// TIA Portal project "Inspection_system" (V16)

(* hardware
DEVICE "S71500/ET200MP station_1"  S7-1500 station
   slot 0: "Rail_0"  Rack  6ES7 590-1***0-0AA0
   slot 1: "PLC_1"  CPU 1515-2 PN  6ES7 515-2AM01-0AB0  V2.8
      slot 3: "CPU display_1"  6ES7591-1BA00-0AA0
      slot 32768: "PROFINET interface_1"  X1
         slot 32769: "Port_1"  X1 P1
         slot 32770: "Port_2"  X1 P2
      slot 33024: "PROFINET interface_2"  X2
         slot 33025: "Port_1"  X2 P1
      slot 34817: "Virtual CP interface port_1"  Virtual CP interface port  Virtual CP interface port
DEVICE "ET 200SP station_1"  ET 200SP-Station
   slot 0: "Rack_0"  Rack  6ES5 710-8MAx1
   slot 0: "IO device_1"  IM 155-6 PN/2 HF  6ES7 155-6AU01-0CN0  V4.2
   slot 1: "AI 4xRTD/TC 2-,3-,4-wire HF_1"  AI 4xRTD/TC 2-,3-,4-wire HF  6ES7 134-6JD00-0CA1  V2.0
      slot 1: "AI 4xRTD/TC 2-,3-,4-wire HF_1"  AI 4xRTD/TC 2-,3-,4-wire HF
   slot 2: "AI 4xRTD/TC 2-,3-,4-wire HF_2"  AI 4xRTD/TC 2-,3-,4-wire HF  6ES7 134-6JD00-0CA1  V2.0
      slot 1: "AI 4xRTD/TC 2-,3-,4-wire HF_2"  AI 4xRTD/TC 2-,3-,4-wire HF
   slot 3: "AI 4xRTD/TC 2-,3-,4-wire HF_3"  AI 4xRTD/TC 2-,3-,4-wire HF  6ES7 134-6JD00-0CA1  V2.0
      slot 1: "AI 4xRTD/TC 2-,3-,4-wire HF_3"  AI 4xRTD/TC 2-,3-,4-wire HF
   slot 4: "AI 8xI 2-,4-wire BA_1"  AI 8xI 2-,4-wire BA  6ES7 134-6GF00-0AA1  V1.0
      slot 1: "AI 8xI 2-,4-wire BA_1"  AI 8xI 2-,4-wire BA
   slot 5: "AQ 4xU/I ST_1"  AQ 4xU/I ST  6ES7 135-6HD00-0BA1  V1.1
      slot 1: "AQ 4xU/I ST_1"  AQ 4xU/I ST
   slot 6: "AQ 4xU/I ST_2"  AQ 4xU/I ST  6ES7 135-6HD00-0BA1  V1.1
      slot 1: "AQ 4xU/I ST_2"  AQ 4xU/I ST
   slot 7: "AQ 4xU/I ST_3"  AQ 4xU/I ST  6ES7 135-6HD00-0BA1  V1.1
      slot 1: "AQ 4xU/I ST_3"  AQ 4xU/I ST
   slot 8: "AQ 4xU/I ST_4"  AQ 4xU/I ST  6ES7 135-6HD00-0BA1  V1.1
      slot 1: "AQ 4xU/I ST_4"  AQ 4xU/I ST
   slot 9: "AQ 4xU/I ST_5"  AQ 4xU/I ST  6ES7 135-6HD00-0BA1  V1.1
      slot 1: "AQ 4xU/I ST_5"  AQ 4xU/I ST
   slot 10: "AQ 4xU/I ST_6"  AQ 4xU/I ST  6ES7 135-6HD00-0BA1  V1.1
      slot 1: "AQ 4xU/I ST_6"  AQ 4xU/I ST
   slot 11: "AQ 4xU/I ST_7"  AQ 4xU/I ST  6ES7 135-6HD00-0BA1  V1.1
      slot 1: "AQ 4xU/I ST_7"  AQ 4xU/I ST
   slot 12: "AQ 4xU/I ST_8"  AQ 4xU/I ST  6ES7 135-6HD00-0BA1  V1.1
      slot 1: "AQ 4xU/I ST_8"  AQ 4xU/I ST
   slot 13: "DI 16x24VDC ST_1"  DI 16x24VDC ST  6ES7 131-6BH01-0BA0  V0.0
      slot 1: "DI 16x24VDC ST_1"  DI 16x24VDC ST
   slot 14: "DQ 16x24VDC/0.5A ST_1"  DQ 16x24VDC/0.5A ST  6ES7 132-6BH01-0BA0  V0.0
      slot 1: "DQ 16x24VDC/0.5A ST_1"  DQ 16x24VDC/0.5A ST
   slot 15: "DQ 16x24VDC/0.5A ST_2"  DQ 16x24VDC/0.5A ST  6ES7 132-6BH01-0BA0  V0.0
      slot 1: "DQ 16x24VDC/0.5A ST_2"  DQ 16x24VDC/0.5A ST
   slot 16: "Server module_1"  Server module  6ES7 193-6PA00-0AA0  V1.1
      slot 1: "Server module_1"  Server module
   slot 127: "BA 2xRJ45"  BA 2xRJ45  6ES7 193-6AR00-0AA0  V0.0
      slot 1: "Port_1"  X1 P1 R  6ES7 193-6AR00-0AA0  V0.0
      slot 2: "Port_2"  X1 P2 R  6ES7 193-6AR00-0AA0  V0.0
*)

// ===== PLC "PLC_1"  CPU 1515-2 PN =====

VAR_GLOBAL   // PLC tag table "Default tag table"
   "upTempLaser1" AT %IW42 : Int;   // (Ain0.0)
   "upTempLaser2" AT %IW44 : Int;   // (Ain0.1)
   "upTempCam1" AT %IW46 : Int;   // (Ain0.2)
   "upTempCam2" AT %IW48 : Int;   // (Ain0.3)
   "downTempLaser1" AT %IW8 : Int;   // (Ain0.4)
   "downTempLaser2" AT %IW10 : Int;   // (Ain0.5)
   "downTempCam1" AT %IW12 : Int;   // (Ain0.6)
   "downTempCam2" AT %IW14 : Int;   // (Ain0.7)
   "airTemperatur" AT %IW16 : Int;   // (Ain1.0)
   "speedRaw" AT %IW24 : Int;   // (Ain2.0)
   "upBlue1" AT %QW0 : Int;
   "upBlue2" AT %QW2 : Int;
   "upBlue3" AT %QW4 : Int;
   "upGreen1" AT %QW6 : Int;
   "upGreen2" AT %QW8 : Int;
   "upGreen3" AT %QW10 : Int;
   "upBlue4" AT %QW12 : Int;
   "upBlue5" AT %QW14 : Int;
   "upBlue6" AT %QW16 : Int;
   "upGreen4" AT %QW18 : Int;
   "upGreen5" AT %QW20 : Int;
   "upGreen6" AT %QW22 : Int;
   "upBlue7" AT %QW24 : Int;
   "upBlue8" AT %QW26 : Int;
   "upBlue9" AT %QW28 : Int;
   "downGreen1" AT %QW32 : Int;
   "downGreen2" AT %QW34 : Int;
   "downGreen3" AT %QW36 : Int;
   "downBlue1" AT %QW38 : Int;
   "downBlue2" AT %QW40 : Int;
   "downBlue3" AT %QW42 : Int;
   "downGreen4" AT %QW44 : Int;
   "downGreen5" AT %QW46 : Int;
   "downGreen6" AT %QW48 : Int;
   "downBlue4" AT %QW50 : Int;
   "downBlue5" AT %QW52 : Int;
   "downBlue6" AT %QW54 : Int;
   "downGreen7" AT %QW56 : Int;
   "downGreen8" AT %QW58 : Int;
   "downGreen9" AT %QW60 : Int;
   "door1" AT %I40.0 : Bool;   // Дверь-1
   "door2" AT %I40.1 : Bool;   // Дверь-2
   "power1_1Ok" AT %I40.2 : Bool;   // Питание внешних цепей
   "power1_2Ok" AT %I40.3 : Bool;   // Питание внутренних цепей
   "laserModeManual" AT %I40.6 : Bool;   // Режим лазеров - Ручной
   "laserModeAuto" AT %I40.7 : Bool;   // Режим лазеров - Автомат
   "veloModeManual" AT %I40.4 : Bool;   // Режим велосиметра - Ручной
   "veloModeAuto" AT %I40.5 : Bool;   // Режим велосиметра - Автомат
   "runForward" AT %I41.0 : Bool;   // Сигнал с цеха -- движение прямо
   "runBackward" AT %I41.1 : Bool;   // Сигнал с цеха -- движение обратно
   "resetAlm" AT %I41.2 : Bool;   // от кнопки сброса аварийного триггера
   "power2_1Ok" AT %I41.3 : Bool;   // Резервированный БП 2_2. Шкаф видеоинспекции, синхробокс и лазеры.
   "power2_2Ok" AT %I41.4 : Bool;   // Резервированный 2_1. Шкаф видеоинспекции, синхробокс и лазеры.
   "upBlue123" AT %Q64.0 : Bool;   // Включение синих лазеров BR1.1-BR1.3. Верх
   "upGreen123" AT %Q64.1 : Bool;   // Включение зелёных лазеров BR2.1-BR2.3. Верх
   "upBlue456" AT %Q64.2 : Bool;   // Включение синих лазеров BR3.1-BR3.3. Верх
   "upGreen456" AT %Q64.3 : Bool;   // Включение зелёных лазеров BR4.1-BR4.3. Верх
   "upBlue789" AT %Q64.4 : Bool;   // Включение синих лазеров BR5.1-BR5.3. Верх
   "downGreen123" AT %Q64.5 : Bool;   // Включение зелёных лазеров BR6.1-BR6.3. Низ
   "downBlue123" AT %Q64.6 : Bool;   // Включение синих лазеров BR7.1-BR7.3. Низ
   "downGreen465" AT %Q64.7 : Bool;   // Включение зелёных лазеров BR8.1-BR8.3. Низ
   "downBlue456" AT %Q65.0 : Bool;   // Включение синих лазеров BR9.1-BR9.3. Низ
   "downGreen789" AT %Q65.1 : Bool;   // Включение зелёных лазеров BR10.1-BR10.3. Низ
   "enLaserVelo" AT %Q66.0 : Bool;   // Лазер велосиметра
   "enGaugeVelo" AT %Q66.1 : Bool;   // Шторка затвора велосиметра
   "airClean" AT %Q66.2 : Bool;   // Клапан воздушного обдува (чистка стекол)
   "runSynchro" AT %Q66.3 : Bool;   // Пуск синхронизации
   "coolUpLaser" AT %Q66.4 : Bool;   // Вентиляторы верхних лазеров
   "coolUpCam" AT %Q66.5 : Bool;   // Вентилятор верхних камер
   "coolDownLaser" AT %Q66.6 : Bool;   // Вентиляторы нижних лазеров
   "coolDownCam" AT %Q66.7 : Bool;   // Вентилятор нижних камер
   "redLamp" AT %Q67.0 : Bool;   // Статус "Работа". Красная лампа.
   "greenLamp" AT %Q67.1 : Bool;   // Статус "Установка отключена". Зелёная лампа.
   "allCooling" AT %Q67.2 : Bool;   // Включение охладителя
   "reverse" AT %Q67.3 : Bool;   // Обратный ход линии
   "Tag_1" AT %M20.0 : Bool;
   "Tag_2" AT %M20.1 : Bool;
   "Tag_3" AT %M20.2 : Bool;
   "System_Byte" AT %MB1 : Byte;
   "FirstScan" AT %M1.0 : Bool;
   "DiagStatusUpdate" AT %M1.1 : Bool;
   "AlwaysTRUE" AT %M1.2 : Bool;
   "AlwaysFALSE" AT %M1.3 : Bool;
   "Clock_Byte" AT %MB0 : Byte;
   "Clock_10Hz" AT %M0.0 : Bool;
   "Clock_5Hz" AT %M0.1 : Bool;
   "Clock_2.5Hz" AT %M0.2 : Bool;
   "Clock_2Hz" AT %M0.3 : Bool;
   "Clock_1.25Hz" AT %M0.4 : Bool;
   "Clock_1Hz" AT %M0.5 : Bool;
   "Clock_0.625Hz" AT %M0.6 : Bool;
   "Clock_0.5Hz" AT %M0.7 : Bool;
END_VAR

DATA_BLOCK "Main_PRG"   // DB4
{ S7_Optimized_Access := 'TRUE' }
VERSION : 0.1
   VAR RETAIN
      AinOffset : Struct
         upTempLaser1 : Real;
         upTempLaser2 : Real;
         upTempCam1 : Real;
         upTempCam2 : Real;
         downTempLaser1 : Real;
         downTempLaser2 : Real;
         downTempCam1 : Real;
         downTempCam2 : Real;
         airTemperatur : Real;
         speed : Real;
      END_STRUCT;
   END_VAR
   VAR
      Ainputs : Struct
         upTempLaser1 : Real;
         upTempLaser2 : Real;
         upTempCam1 : Real;
         upTempCam2 : Real;
         downTempLaser1 : Real;
         downTempLaser2 : Real;
         downTempCam1 : Real;
         downTempCam2 : Real;
         airTemperatur : Real;
         speed : Real;
      END_STRUCT;
      fault_buffer : Struct   // 64bit -- Биты аварий
         door1 : Bool;   // Дверь1 -- открыта
         door2 : Bool;   // Дверь2 -- открыта
         power11 : Bool;   // Питание внешних цепей
         power12 : Bool;   // Питание внутренних цепей
         power2 : Bool;   // Питание лазеров, ШВИ, синхробокса, видеокамер
         upLaserTemp : Bool;   // Температура выше аварийного уровня. (Верхний блок лазеров)
         upLaserAllCh : Bool;   // Все каналы измерения температуры неисправны. (Верхний блок лазеров)
         upCamTemp : Bool;   // Температура выше аварийного уровня. (Верхний блок камер)
         upCamAllCh : Bool;   // Все каналы измерения температуры неисправны. (Верхний блок камер)
         downLaserTemp : Bool;   // Температура выше аварийного уровня. (Нижний блок лазеров)
         downLaserAllCh : Bool;   // Все каналы измерения температуры неисправны. (Нижний блок лазеров)
         downCamTemp : Bool;   // Температура выше аварийного уровня. (Нижний блок камер)
         downCamAllCh : Bool;   // Все каналы измерения температуры неисправны. (Нижний блок камер)
         Ain2MinLimit : Bool;   // Вход от велосиметра (4-20мА) ниже уровня 4мА
         Ain2MaxLimit : Bool;   // Вход от велосиметра (4-20мА) выше уровня 20мА
         iniError : Bool;   // Ошибка инициализации.
         gaugeOk : Bool;
         lasTempH : Bool := false;
         lasTempL : Bool := false;
         caseTempH : Bool := false;
         caseTempL : Bool := false;
         gaugeH : Bool := false;
         veloNoConnect : Bool;
         reserve7 : Bool := false;
         reserve8 : Bool := false;
         reserve9 : Bool := false;
         reserve10 : Bool := false;
         reserve11 : Bool := false;
         reserve12 : Bool := false;
         reserve13 : Bool := false;
         reserve14 : Bool := false;
         reserve15 : Bool := false;
         reserve16 : Bool := false;
         reserve17 : Bool := false;
         reserve18 : Bool := false;
         reserve19 : Bool := false;
         reserve20 : Bool := false;
         reserve21 : Bool := false;
         reserve22 : Bool := false;
         reserve23 : Bool := false;
         reserve24 : Bool := false;
         reserve25 : Bool := false;
         reserve26 : Bool := false;
         reserve27 : Bool := false;
         reserve28 : Bool := false;
         reserve29 : Bool := false;
         reserve30 : Bool := false;
         reserve31 : Bool := false;
      END_STRUCT;
      iniOk : Bool;
      initializing : Bool;
      RUN : Bool;
      errUpTempLaser1 : Bool;   // (Ain0.0)
      errUpTempLaser2 : Bool;   // (Ain0.1)
      errUpTempCam1 : Bool;   // (Ain0.2)
      errUpTempCam2 : Bool;   // (Ain0.3)
      errDownTempLaser1 : Bool;   // (Ain0.4)
      errDownTempLaser2 : Bool;   // (Ain0.5)
      errDownTempCam1 : Bool;   // (Ain0.6)
      errDownTempCam2 : Bool;   // (Ain0.7)
      errAirTemperatur : Bool;   // (Ain1.0)
      synchroOn : Bool;
      t0 : Bool;
      t1 : Bool := false;
      t2 : Bool := false;
      t3 : Bool := false;
      t4 : Bool := false;
      t5 : Bool := false;
      configAI0 : Struct
         modulInfo0 : Byte;   // версия
         modulInfo1 : Byte;   // Количество структур следующих параметров
         modulInfo2 : Byte;   // Количество следующих блоков параметров модуля
         modulInfo3 : Byte;   // длина блока параметров модуля
         modulParam4 : Byte;   // bit0 -- Отсутствует напряжение питания.
         modulParam5 : Byte := 16#0;   // резерв
         modulParam6 : Byte := 16#0;
         modulParam7 : Byte := 16#0;
         modulParam8 : Byte := 16#0;
         modulParam9 : Byte := 16#0;
         channelInfo10 : Byte;   // количество следующих блоков параметров канала
         channelInfo11 : Byte := 16#0;   // Длина блока параметров канала
         "0channel0_12" : Byte;   // Тип измерения
         "1channel0_13" : Byte := 16#0;   // Диапазон измерений
         "2channel0_14" : Byte := 16#0;   // Температурный коэффициент
         "3channel0_15" : Byte := 16#0;   // Сглаживание
         "4channel0_16" : Byte := 16#0;   // Единица измерения и тип подключения
         "5channel0_17" : Byte := 16#0;   // бит4 - превышен лимит2, бит5 - ниже лимита2, бит6 - превышен лимит1, бит7 - ниже лимита1
         "6channel0_18" : Byte := 16#0;   // бит1-общий режим, бит2-короткое замыкание, бит4-обрыв, бит5-компенсация, бит6-ниже, бит7-выше
         "7channel0_19" : Byte := 16#0;   // резерв
         "8channel0_20" : Byte := 16#0;   // резерв
         "9channel0_21" : Byte := 16#0;   // резерв
         "10channel0_22" : Byte := 16#0;   // hardware interrupt1, high limit, byte0
         "11channel0_23" : Byte := 16#0;   // hardware interrupt1, high limit, byte1
         "12channel0_24" : Byte := 16#0;   // hardware interrupt1, low limit, byte0
         "13channel0_25" : Byte := 16#0;   // hardware interrupt1, low limit, byte1
         "14channel0_26" : Byte := 16#0;   // hardware interrupt2, high limit, byte0
         "15channel0_27" : Byte := 16#0;   // hardware interrupt2, high limit, byte1
         "16channel0_28" : Byte := 16#0;   // hardware interrupt2, low limit, byte0
         "17channel0_29" : Byte := 16#0;   // hardware interrupt2, low limit, byte1
         "18channel0_30" : Byte := 16#0;   // сопротивление, byte0
         "19channel0_31" : Byte := 16#0;   // сопротивление, byte1
         "20channel0_32" : Byte := 16#0;   // резерв
         "21channel0_33" : Byte := 16#0;   // резерв
         "0channel1_34" : Byte := 16#0;   // Тип измерения
         "1channel1_35" : Byte := 16#0;   // Диапазон измерений
         "2channel1_36" : Byte := 16#0;   // Температурный коэффициент
         "3channel1_37" : Byte := 16#0;   // Сглаживание
         "4channel1_38" : Byte := 16#0;   // Единица измерения и тип подключения
         "5channel1_39" : Byte := 16#0;   // бит4 - превышен лимит2, бит5 - ниже лимита2, бит6 - превышен лимит1, бит7 - ниже лимита1
         "6channel1_40" : Byte := 16#0;   // бит1-общий режим, бит2-короткое замыкание, бит4-обрыв, бит5-компенсация, бит6-ниже, бит7-выше
         "7channel1_41" : Byte := 16#0;   // резерв
         "8channel1_42" : Byte := 16#0;   // резерв
         "9channel1_43" : Byte := 16#0;   // резерв
         "10channel1_44" : Byte := 16#0;   // hardware interrupt1, high limit, byte0
         "11channel1_45" : Byte := 16#0;   // hardware interrupt1, high limit, byte1
         "12channel1_46" : Byte := 16#0;   // hardware interrupt1, low limit, byte0
         "13channel1_47" : Byte := 16#0;   // hardware interrupt1, low limit, byte1
         "14channel1_48" : Byte := 16#0;   // hardware interrupt2, high limit, byte0
         "15channel1_49" : Byte := 16#0;   // hardware interrupt2, high limit, byte1
         "16channel1_50" : Byte := 16#0;   // hardware interrupt2, low limit, byte0
         "17channel1_51" : Byte := 16#0;   // hardware interrupt2, low limit, byte1
         "18channel1_52" : Byte := 16#0;   // сопротивление, byte0
         "19channel1_53" : Byte := 16#0;   // сопротивление, byte1
         "20channel1_54" : Byte := 16#0;   // резерв
         "21channel1_55" : Byte := 16#0;   // резерв
         "0channel2_56" : Byte := 16#0;   // Тип измерения
         "1channel2_57" : Byte := 16#0;   // Диапазон измерений
         "2channel2_58" : Byte := 16#0;   // Температурный коэффициент
         "3channel2_59" : Byte := 16#0;   // Сглаживание
         "4channel2_60" : Byte := 16#0;   // Единица измерения и тип подключения
         "5channel2_61" : Byte := 16#0;   // бит4 - превышен лимит2, бит5 - ниже лимита2, бит6 - превышен лимит1, бит7 - ниже лимита1
         "6channel2_62" : Byte := 16#0;   // бит1-общий режим, бит2-короткое замыкание, бит4-обрыв, бит5-компенсация, бит6-ниже, бит7-выше
         "7channel2_63" : Byte := 16#0;   // резерв
         "8channel2_64" : Byte := 16#0;   // резерв
         "9channel2_65" : Byte := 16#0;   // резерв
         "10channel2_66" : Byte := 16#0;   // hardware interrupt1, high limit, byte0
         "11channel2_67" : Byte := 16#0;   // hardware interrupt1, high limit, byte1
         "12channel2_68" : Byte := 16#0;   // hardware interrupt1, low limit, byte0
         "13channel2_69" : Byte := 16#0;   // hardware interrupt1, low limit, byte1
         "14channel2_70" : Byte := 16#0;   // hardware interrupt2, high limit, byte0
         "15channel2_71" : Byte := 16#0;   // hardware interrupt2, high limit, byte1
         "16channel2_72" : Byte := 16#0;   // hardware interrupt2, low limit, byte0
         "17channel2_73" : Byte := 16#0;   // hardware interrupt2, low limit, byte1
         "18channel2_74" : Byte := 16#0;   // сопротивление, byte0
         "19channel2_75" : Byte := 16#0;   // сопротивление, byte1
         "20channel2_76" : Byte := 16#0;   // резерв
         "21channel2_77" : Byte := 16#0;   // резерв
         "0channel3_78" : Byte := 16#0;   // Тип измерения
         "1channel3_79" : Byte := 16#0;   // Диапазон измерений
         "2channel3_80" : Byte := 16#0;   // Температурный коэффициент
         "3channel3_81" : Byte := 16#0;   // Сглаживание
         "4channel3_82" : Byte := 16#0;   // Единица измерения и тип подключения
         "5channel3_83" : Byte := 16#0;   // бит4 - превышен лимит2, бит5 - ниже лимита2, бит6 - превышен лимит1, бит7 - ниже лимита1
         "6channel3_84" : Byte := 16#0;   // бит1-общий режим, бит2-короткое замыкание, бит4-обрыв, бит5-компенсация, бит6-ниже, бит7-выше
         "7channel3_85" : Byte := 16#0;   // резерв
         "8channel3_86" : Byte := 16#0;   // резерв
         "9channel3_87" : Byte := 16#0;   // резерв
         "10channel3_88" : Byte := 16#0;   // hardware interrupt1, high limit, byte0
         "11channel3_89" : Byte := 16#0;   // hardware interrupt1, high limit, byte1
         "12channel3_90" : Byte := 16#0;   // hardware interrupt1, low limit, byte0
         "13channel3_91" : Byte := 16#0;   // hardware interrupt1, low limit, byte1
         "14channel3_92" : Byte := 16#0;   // hardware interrupt2, high limit, byte0
         "15channel3_93" : Byte := 16#0;   // hardware interrupt2, high limit, byte1
         "16channel3_94" : Byte := 16#0;   // hardware interrupt2, low limit, byte0
         "17channel3_95" : Byte := 16#0;   // hardware interrupt2, low limit, byte1
         "18channel3_96" : Byte := 16#0;   // сопротивление, byte0
         "19channel3_97" : Byte := 16#0;   // сопротивление, byte1
         "20channel3_98" : Byte := 16#0;   // резерв
         "21channel3_99" : Byte := 16#0;   // резерв
      END_STRUCT;
   END_VAR
BEGIN
END_DATA_BLOCK

DATA_BLOCK "READ"   // DB200
{ S7_Optimized_Access := 'FALSE' }
VERSION : 0.1
   VAR
      fault : Struct   // 64bit -- Биты аварий
         door1 : Bool;   // Дверь1 -- открыта
         door2 : Bool;   // Дверь2 -- открыта
         power11 : Bool;   // Питание внешних цепей
         power12 : Bool;   // Питание внутренних цепей
         power2 : Bool;   // Питание лазеров, ШВИ, синхробокса, видеокамер
         upLaserTemp : Bool;   // Температура выше аварийного уровня. (Верхний блок лазеров)
         upLaserAllCh : Bool;   // Все каналы измерения температуры неисправны. (Верхний блок лазеров)
         upCamTemp : Bool;   // Температура выше аварийного уровня. (Верхний блок камер)
         upCamAllCh : Bool;   // Все каналы измерения температуры неисправны. (Верхний блок камер)
         downLaserTemp : Bool;   // Температура выше аварийного уровня. (Нижний блок лазеров)
         downLaserAllCh : Bool;   // Все каналы измерения температуры неисправны. (Нижний блок лазеров)
         downCamTemp : Bool;   // Температура выше аварийного уровня. (Нижний блок камер)
         downCamAllCh : Bool;   // Все каналы измерения температуры неисправны. (Нижний блок камер)
         Ain2MinLimit : Bool;   // Вход от велосиметра (4-20мА) ниже уровня 4мА
         Ain2MaxLimit : Bool;   // Вход от велосиметра (4-20мА) выше уровня 20мА
         iniError : Bool;   // Ошибка инициализации.
         gaugeOk : Bool;   // Неисправность измерителя велосиметра
         lasTempH : Bool := false;   // Высокая температура лазера велосиметра
         lasTempL : Bool := false;   // Низкая температура лазера велосиметра
         caseTempH : Bool := false;   // Высокая температура корпуса велосиметра
         caseTempL : Bool := false;   // Низкая температура корпуса велосиметра
         gaugeH : Bool := false;   // Перегрев измерителя велосиметра
         veloNoConnect : Bool;   // Отсутствует соединение с велосиметром
         reserve7 : Bool := false;
         reserve8 : Bool := false;
         reserve9 : Bool := false;
         reserve10 : Bool := false;
         reserve11 : Bool := false;
         reserve12 : Bool := false;
         reserve13 : Bool := false;
         reserve14 : Bool := false;
         reserve15 : Bool := false;
         reserve16 : Bool := false;
         reserve17 : Bool := false;
         reserve18 : Bool := false;
         reserve19 : Bool := false;
         reserve20 : Bool := false;
         reserve21 : Bool := false;
         reserve22 : Bool := false;
         reserve23 : Bool := false;
         reserve24 : Bool := false;
         reserve25 : Bool := false;
         reserve26 : Bool := false;
         reserve27 : Bool := false;
         reserve28 : Bool := false;
         reserve29 : Bool := false;
         reserve30 : Bool := false;
         reserve31 : Bool := false;
      END_STRUCT;
      warning : Struct   // 96bit -- Биты предупреждений
         highTempUpLaser : Bool;   // Температура выше warning уровня. (Верхний блок лазеров)
         highTempUpCam : Bool;   // Температура выше warning уровня. (Верхний блок камер)
         highTempDownLaser : Bool;   // Температура выше warning уровня. (Нижний блок лазеров)
         highTempDownCam : Bool;   // Температура выше warning уровня. (Нижний блок камер)
         highTempPneumatic : Bool;   // Температура выше аварийного уровня. (Воздуха в пневмосистеме)
         power2_1 : Bool;   // Резервированный БП-1 неисправен. (Питание лазеров, ШВИ, синхробокса, видеокамер)
         power2_2 : Bool := false;   // Резервированный БП-2 неисправен. (Питание лазеров, ШВИ, синхробокса, видеокамер)
         overFlowUpLaserAin00 : Bool := false;   // Сопротивление датчика 1 температуры выше допустимого (Верхний блок лазеров)
         overFlowUpLaserAin01 : Bool := false;   // Сопротивление датчика 2 температуры выше допустимого (Верхний блок лазеров)
         overFlowUpCamAin02 : Bool := false;   // Сопротивление датчика 1 температуры выше допустимого (Верхний блок камер)
         overFlowUpCamAin03 : Bool := false;   // Сопротивление датчика 2 температуры выше допустимого (Верхний блок камер)
         overFlowDownLaserAin04 : Bool := false;   // Сопротивление датчика 1 температуры выше допустимого (Нижний блок лазеров)
         overFlowDownLaserAin05 : Bool := false;   // Сопротивление датчика 2 температуры выше допустимого (Нижний блок лазеров)
         overFlowDownCamAin06 : Bool := false;   // Сопротивление датчика 1 температуры выше допустимого (Нижний блок камер)
         overFlowDownCamAin07 : Bool := false;   // Сопротивление датчика 2 температуры выше допустимого (Нижний блок камер)
         overFlowPneumaticAin10 : Bool := false;   // Сопротивление датчика температуры выше допустимого (Воздух в пневмосистеме)
         underFlowUpLaserAin00 : Bool := false;   // Сопротивление датчика 1 температуры ниже допустимого (Верхний блок лазеров)
         underFlowUpLaserAin01 : Bool := false;   // Сопротивление датчика 2 температуры ниже допустимого (Верхний блок лазеров)
         underFlowUpCamAin02 : Bool := false;   // Сопротивление датчика 1 температуры ниже допустимого (Верхний блок камер)
         underFlowUpCamAin03 : Bool := false;   // Сопротивление датчика 2 температуры ниже допустимого (Верхний блок камер)
         underFlowDownLaserAin04 : Bool := false;   // Сопротивление датчика 1 температуры ниже допустимого (Нижний блок лазеров)
         underFlowDownLaserAin05 : Bool := false;   // Сопротивление датчика 2 температуры ниже допустимого (Нижний блок лазеров)
         underFlowDownCamAin06 : Bool := false;   // Сопротивление датчика 1 температуры ниже допустимого (Нижний блок камер)
         underFlowDownCamAin07 : Bool := false;   // Сопротивление датчика 2 температуры ниже допустимого (Нижний блок камер)
         underFlowPneumaticAin10 : Bool := false;   // Сопротивление датчика температуры ниже допустимого (Воздух в пневмосистеме)
         reserve6 : Bool := false;
         reserve5 : Bool := false;
         reserve4 : Bool := false;
         reserve3 : Bool := false;
         reserve2 : Bool := false;
         reserve1 : Bool := false;
         reserve0 : Bool := false;
      END_STRUCT;
      velometer : Struct
         dw0 : Struct
            measMode : Bool;   // Measurement mode. 0=Normal;1=Batch
            resolut : Bool := false;   // Resolution of length output. 0=length 0.0001;1=length 0.1
            speedResp : Bool := false;   // Speed reponse for pulse and analogue output. 0=Instant;1=Averaged
            b3 : Bool := false;
            b4 : Bool := false;
            b5 : Bool := false;
            b6 : Bool := false;
            b7 : Bool := false;
            measLen1 : Bool := false;   // 1=>Preset
            measLen2 : Bool := false;   // 1=>Preset
            b10 : Bool := false;
            laserOn : Bool := false;   // 1= ON;0=OFF
            readingSpeed : Bool := false;   // 1=Valid;0=Invalid
            objectDetect : Bool := false;   // 1=Object detected;0=No object
            reading : Bool := false;   // Good reading status. 1=Lower than threshold;0=OK
            b15 : Bool := false;
         END_STRUCT;
         dw1 : Struct
            gaugeOk : Bool;   // 1=OK;0=Failed
            lasTempH : Bool := false;   // Laser temperature too high. 1=Too high;0=OK
            lasTempL : Bool := false;   // Laser temperature too low. 1=Too low;0=OK
            caseTempH : Bool := false;   // Case temperature too high. 1=Too low;0=OK
            caseTempL : Bool := false;   // Case temperature too low. 1=Too low;0=OK
            reflectionH : Bool := false;   // Light reflection too strong. 1=Too low;0=OK
            gaugeH : Bool := false;   // Gauge too hot. 1=Too low;0=OK
            b7 : Bool := false;
            b8 : Bool := false;
            b9 : Bool := false;
            b10 : Bool := false;
            b11 : Bool := false;
            b12 : Bool := false;
            b13 : Bool := false;
            b14 : Bool := false;
            b15 : Bool := false;
         END_STRUCT;
         averSpeed : Real;   // Отфильтрованная скорость
         instSpeed : Real;   // Мгновенная скорость
         totalLen : Real;   // Общая длина
         batchLen : Real;   // длина партии
         lastLen : Real;   // предыдущая сохраненная длина
         reelNum : DInt;   // номер измерения
         batchNum : Int;   // 0~65535
         readingLavel : Int;   // 0~100%. Качество фокуса и отраженного сигнала
         SNR : Int;   // 0~65535
         SLX : Int;   // ±200mm
      END_STRUCT;
      inputs : Struct   // 16bit -- Дискретные входы
         door1 : Bool;   // Дверь-1
         door2 : Bool;   // Дверь-2
         power1_1Ok : Bool;   // Питание внешних цепей
         power1_2Ok : Bool;   // Питание внутренних цепей
         laserModeManual : Bool;   // Режим лазеров - Ручной
         laserModeAuto : Bool;   // Режим лазеров - Автомат
         veloModeManual : Bool;   // Режим велосиметра - Ручной
         veloModeAuto : Bool;   // Режим велосиметра - Автомат
         runForward : Bool;   // Сигнал с цеха -- движение прямо
         runBackward : Bool;   // Сигнал с цеха -- движение обратно
         resetAlm : Bool;   // от кнопки сброса аварийного триггера
         power2_1Ok : Bool;   // Резервированный БП 2_2. Шкаф видеоинспекции, синхробокс и лазеры.
         power2_2Ok : Bool;   // Резервированный 2_1. Шкаф видеоинспекции, синхробокс и лазеры.
         reserv0 : Bool;
         reserv1 : Bool;
         reserv2 : Bool;
      END_STRUCT;
      outputs : Struct   // 32bit -- Дискретные входы
         upBlue123 : Bool;   // Включение синих лазеров BR1.1-BR1.3. Верх
         upGreen123 : Bool;   // Включение зелёных лазеров BR2.1-BR2.3. Верх
         upBlue456 : Bool;   // Включение синих лазеров BR3.1-BR3.3. Верх
         upGreen456 : Bool;   // Включение зелёных лазеров BR4.1-BR4.3. Верх
         upBlue789 : Bool;   // Включение синих лазеров BR5.1-BR5.3. Верх
         downGreen123 : Bool;   // Включение зелёных лазеров BR6.1-BR6.3. Низ
         downBlue123 : Bool;   // Включение синих лазеров BR7.1-BR7.3. Низ
         downGreen465 : Bool;   // Включение зелёных лазеров BR8.1-BR8.3. Низ
         downBlue456 : Bool;   // Включение синих лазеров BR9.1-BR9.3. Низ
         downGreen789 : Bool;   // Включение зелёных лазеров BR10.1-BR10.3. Низ
         reserve0 : Bool;
         reserve1 : Bool;
         reserve2 : Bool;
         reserve3 : Bool;
         reserve4 : Bool;
         reserve5 : Bool;
         disVelocimeter : Bool;   // Вкл. лазера велосиметра - True
         enVelocimeter : Bool;   // Вкл. затвора велосиметра - True
         airClean : Bool;   // Клапан воздушного обдува (чистка стекол)
         synchro : Bool;   // Дезактивация синхронизации
         coolUpLaser : Bool;   // Вентиляторы верхних лазеров
         coolUpCam : Bool;   // Вентилятор верхних камер
         coolDownLaser : Bool;   // Вентиляторы нижних лазеров
         coolDownCam : Bool;   // Вентилятор нижних камер
         redLamp : Bool;   // Статус "Работа". Красная лампа.
         greenLamp : Bool;   // Статус "Установка отключена". Зелёная лампа.
         airCooller : Bool;   // Включение охладителя
         setBackward : Bool;   // Обратный ход линии (незадействован)
         reserve6 : Bool;
         reserve7 : Bool;
         reserve8 : Bool;
         reserve9 : Bool;
      END_STRUCT;
      status : Struct
         redLamp : Bool;   // Постоянно true -- Работа. Mигание -- авария.
         greenLamp : Bool;   // Постоянно true -- инциализация пройдена, готовность к включению.
         airCooller : Bool;   // Охладитель воздуха
         veloPositive : Bool;   // Линия движется прямо
         veloNegative : Bool;   // Линия движется обратно
         warning : Bool;   // Наличие предупреждения
         errorTrigg : Bool;   // флаг наличия предупреждения
         reserv0 : Bool;   // флаг триггера аварии
         reserv1 : Bool;
         reserv2 : Bool;
         reserv3 : Bool;
         reserv4 : Bool;
         reserv5 : Bool;
         reserv6 : Bool;
         reserv7 : Bool;
         reserv8 : Bool := false;
         statusCode : Int;   // (+10 -- Предупреждение). 0 -- ожидание; 1 -- инициализация; 2 -- Готовность; 3 -- Работа(режим Авто); 4 -- Работа(руч. режим); 5 -- Авария.
         reservInt0 : Int;
         reservInt1 : Int := 0;
      END_STRUCT;
      temperatures : Struct
         upLaserTemp : Real;   // Текущая температура. (Верхний блок лазеров)
         upCamTemp : Real;   // Текущая температура. (Верхний блок камер)
         downLaserTemp : Real;   // Текущая температура. (Нижний блок лазеров)
         downCamTemp : Real;   // Текущая температура. (Нижний блок камер)
         pneumaticTemp : Real;   // Текущая температура. (Воздуха в пневмосистеме)
         reserv0 : Real;
         reserv1 : Real := 0.0;
      END_STRUCT;
      dbWrite : Struct
         resetErrorTrigg : Bool;   // Сброс аварии
         coolAirEn : Bool;
         setLasersManual : Struct   // Для ручного режима
            upBlueLasers123 : Bool := false;
            upGreenLasers123 : Bool := false;
            upBlueLasers456 : Bool := false;
            upGreenLasers456 : Bool := false;
            upBlueLasers789 : Bool := false;
            downGreenLasers123 : Bool := false;
            downBlueLasers123 : Bool := false;
            downGreenLasers465 : Bool := false;
            downBlueLasers456 : Bool := false;
            downGreenLasers789 : Bool := false;
         END_STRUCT;
         simulate : Struct   // Симуляция каналов. (для АО применимо из setPowerLasers)
            DI : Struct
               DI0 : USInt := 16#0;
               DI1 : USInt := 16#0;
               DI2 : USInt := 16#0;
               DI3 : USInt := 16#0;
               DI4 : USInt := 16#0;
               DI5 : USInt := 16#0;
               DI6 : USInt := 16#0;
               DI7 : USInt := 16#0;
               DI8 : USInt := 16#0;
               DI9 : USInt := 16#0;
               DI10 : USInt := 16#0;
               DI11 : USInt := 16#0;
               DI12 : USInt := 16#0;
               DI13 : USInt := 16#0;
               DI14 : USInt := 16#0;
               DI15 : USInt := 16#0;
            END_STRUCT;
            "DO" : Struct
               DO0 : USInt := 0;
               DO1 : USInt := 0;
               DO2 : USInt := 0;
               DO3 : USInt := 0;
               DO4 : USInt := 0;
               DO5 : USInt := 0;
               DO6 : USInt := 0;
               DO7 : USInt := 0;
               DO8 : USInt := 0;
               DO9 : USInt := 0;
               DO10 : USInt := 0;
               DO11 : USInt := 0;
               DO12 : USInt := 0;
               DO13 : USInt := 0;
               DO14 : USInt := 0;
               DO15 : USInt := 0;
               DO16 : USInt := 0;
               DO17 : USInt := 0;
               DO18 : USInt := 0;
               DO19 : USInt := 0;
               DO20 : USInt := 0;
               DO21 : USInt := 0;
               DO22 : USInt := 0;
               DO23 : USInt := 0;
               DO24 : USInt := 0;
               DO25 : USInt := 0;
               DO26 : USInt := 0;
               DO27 : USInt := 0;
               DO28 : USInt := 0;
               DO29 : USInt := 0;
               DO30 : USInt := 0;
               DO31 : USInt := 0;
            END_STRUCT;
            AI : Struct   // 0.0 -- симуляция отключена; от 0.0 до 0.001 -- запись 0.0; выше 0.001 -- запись любого числа.
               upTempLaser1 : Real := 0.0;
               upTempLaser2 : Real := 0.0;
               upTempCam1 : Real := 0.0;
               upTempCam2 : Real := 0.0;
               downTempLaser1 : Real := 0.0;
               downTempLaser2 : Real := 0.0;
               downTempCam1 : Real := 0.0;
               downTempCam2 : Real := 0.0;
               airTemperatur : Real := 0.0;
               reserv : Real := 0.0;
            END_STRUCT;
         END_STRUCT;
         setTemperatures : Struct   // Уставки температур
            faultUpLaser : Real := 60.0;   // Аварийная температура (по умолч. 60)
            faultUpCam : Real := 60.0;
            faultDownLaser : Real := 60.0;
            faultDownCam : Real := 60.0;
            warnAir : Real := 60.0;   // Предупреждающая температура (по умолч. 60)
            warnUpLaser : Real := 45.0;   // Предупреждающая температура (по умолч. 45)
            warnUpCam : Real := 45.0;   // Предупреждающая температура (по умолч. 45)
            warnDownLaser : Real := 45.0;   // Предупреждающая температура (по умолч. 45)
            warnDownCam : Real := 45.0;   // Предупреждающая температура (по умолч. 45)
            reserv0 : Real;
         END_STRUCT;
         cleanTime : Struct   // Периодичность продувки
            tOnS : Real := 5.0;
            tOffMin : Real := 30.0;
         END_STRUCT;
         setPowerLasers : Struct   // Мощность лазеров (0 -- 100%)
            writeAll : Real := 25.0;
            upBlue1 : Real := 25.0;   // AO0.0
            upBlue2 : Real := 25.0;   // AO0.1
            upBlue3 : Real := 25.0;   // AO0.2
            upGreen1 : Real := 25.0;   // AO0.3
            upGreen2 : Real := 25.0;   // AO0.4
            upGreen3 : Real := 25.0;   // AO0.5
            upBlue4 : Real := 25.0;   // AO0.6
            upBlue5 : Real := 25.0;   // AO0.7
            upBlue6 : Real := 25.0;   // AO1.0
            upGreen4 : Real := 25.0;   // AO1.1
            upGreen5 : Real := 25.0;   // AO1.2
            upGreen6 : Real := 25.0;   // AO1.3
            upBlue7 : Real := 25.0;   // AO1.4
            upBlue8 : Real := 25.0;   // AO1.5
            upBlue9 : Real := 25.0;   // AO1.6
            downGreen1 : Real := 25.0;   // AO2.0
            downGreen2 : Real := 25.0;   // AO2.1
            downGreen3 : Real := 25.0;   // AO2.2
            downBlue1 : Real := 25.0;   // AO2.3
            downBlue2 : Real := 25.0;   // AO2.4
            downBlue3 : Real := 25.0;   // AO2.5
            downGreen4 : Real := 25.0;   // AO2.6
            downGreen5 : Real := 25.0;   // AO2.7
            downGreen6 : Real := 25.0;   // AO3.0
            downBlue4 : Real := 25.0;   // AO3.1
            downBlue5 : Real := 25.0;   // AO3.2
            downBlue6 : Real := 25.0;   // AO3.3
            downGreen7 : Real := 25.0;   // AO3.4
            downGreen8 : Real := 25.0;   // AO3.5
            downGreen9 : Real := 25.0;   // AO3.6
         END_STRUCT;
      END_STRUCT;
   END_VAR
BEGIN
END_DATA_BLOCK

DATA_BLOCK "WRITE"   // DB201
{ S7_Optimized_Access := 'FALSE' }
VERSION : 0.1
   VAR
      resetErrorTrigg : Bool := false;   // Сброс аварии
      coolAirEn : Bool := false;   // Охладитель пневмосистемы
      setLasersManual : Struct   // Для ручного режима
         upBlueLasers123 : Bool := true;   // Питание верхних синих лазеров 1, 2 и 3: ***____________
         upGreenLasers123 : Bool := true;   // Питание верхних зеленые лазеров 1, 2 и 3: ___***_________
         upBlueLasers456 : Bool := true;   // Питание верхних синих лазеров 4, 5 и 6: ______***______
         upGreenLasers456 : Bool := true;   // Питание верхних зеленых лазеров 4, 5 и 6: _________***___
         upBlueLasers789 : Bool := true;   // Питание верхних синих лазеров 7, 8 и 9: ____________***
         downGreenLasers123 : Bool := true;   // Питание нижних зеленых лазеров 1, 2 и 3: ***____________
         downBlueLasers123 : Bool := true;   // Питание нижних синих лазеров 1, 2 и 3: ___***_________
         downGreenLasers465 : Bool := true;   // Питание нижних зеленых лазеров 4, 5 и 6: ______***______
         downBlueLasers456 : Bool := true;   // Питание нижних синих лазеров 4, 5 и 6: _________***___
         downGreenLasers789 : Bool := true;   // Питание нижних зеленых лазеров 7, 8 и 9: ____________***
      END_STRUCT;
      simulate : Struct   // Симуляция каналов. (для АО применимо из setPowerLasers)
         DI : Struct
            DI0 : USInt := 16#0;   // Дверь-1
            DI1 : USInt := 16#0;   // Дверь-2
            DI2 : USInt := 16#0;   // Питание внешних цепей
            DI3 : USInt := 16#0;   // Питание внутренних цепей
            DI4 : USInt := 16#0;   // Режим лазеров - Ручной
            DI5 : USInt := 16#0;   // Режим лазеров - Автомат
            DI6 : USInt := 16#0;   // Режим велосиметра - Ручной
            DI7 : USInt := 16#0;   // Режим велосиметра - Автомат
            DI8 : USInt := 16#0;   // Сигнал с цеха -- движение прямо
            DI9 : USInt := 16#0;   // Сигнал с цеха -- движение обратно
            DI10 : USInt := 16#0;   // от кнопки сброса аварийного триггера
            DI11 : USInt := 16#0;   // Резервированный БП 2_2. Шкаф видеоинспекции, синхробокс и лазеры.
            DI12 : USInt := 16#0;   // Резервированный 2_1. Шкаф видеоинспекции, синхробокс и лазеры.
            DI13 : USInt := 16#0;
            DI14 : USInt := 16#0;
            DI15 : USInt := 16#0;
         END_STRUCT;
         "DO" : Struct
            DO0 : USInt := 0;   // Включение синих лазеров BR1.1-BR1.3. Верх
            DO1 : USInt := 0;   // Включение зелёных лазеров BR2.1-BR2.3. Верх
            DO2 : USInt := 0;   // Включение синих лазеров BR3.1-BR3.3. Верх
            DO3 : USInt := 0;   // Включение зелёных лазеров BR4.1-BR4.3. Верх
            DO4 : USInt := 0;   // Включение синих лазеров BR5.1-BR5.3. Верх
            DO5 : USInt := 0;   // Включение зелёных лазеров BR6.1-BR6.3. Низ
            DO6 : USInt := 0;   // Включение синих лазеров BR7.1-BR7.3. Низ
            DO7 : USInt := 0;   // Включение зелёных лазеров BR8.1-BR8.3. Низ
            DO8 : USInt := 0;   // Включение синих лазеров BR9.1-BR9.3. Низ
            DO9 : USInt := 0;   // Включение зелёных лазеров BR10.1-BR10.3. Низ
            DO10 : USInt := 0;   // Лазер велосиметра
            DO11 : USInt := 0;   // открытие створки (затвора)
            DO12 : USInt := 0;   // Клапан воздушного обдува (чистка стекол)
            DO13 : USInt := 0;   // Пуск синхронизации
            DO14 : USInt := 0;   // Вентиляторы верхних лазеров
            DO15 : USInt := 0;   // Вентилятор верхних камер
            DO16 : USInt := 0;   // Вентиляторы нижних лазеров
            DO17 : USInt := 0;   // Вентилятор нижних камер
            DO18 : USInt := 0;   // Статус "Работа". Красная лампа.
            DO19 : USInt := 0;   // Статус "Установка отключена". Зелёная лампа.
            DO20 : USInt := 0;   // Включение охладителя
            DO21 : USInt := 0;   // Обратный ход линии
            DO22 : USInt := 0;
            DO23 : USInt := 0;
            DO24 : USInt := 0;
            DO25 : USInt := 0;
            DO26 : USInt := 0;
            DO27 : USInt := 0;
            DO28 : USInt := 0;
            DO29 : USInt := 0;
            DO30 : USInt := 0;
            DO31 : USInt := 0;
         END_STRUCT;
         AI : Struct   // 0.0 -- симуляция отключена; от 0.0 до 0.001 -- запись 0.0; выше 0.001 -- запись любого числа.
            upTempLaser1 : Real := 0.0;
            upTempLaser2 : Real := 0.0;
            upTempCam1 : Real := 0.0;
            upTempCam2 : Real := 0.0;
            downTempLaser1 : Real := 0.0;
            downTempLaser2 : Real := 0.0;
            downTempCam1 : Real := 0.0;
            downTempCam2 : Real := 0.0;
            airTemperatur : Real := 0.0;
            reserv : Real := 0.0;
         END_STRUCT;
      END_STRUCT;
      setTemperatures : Struct   // Уставки температур
         faultUpLaser : Real := 45.0;   // Уставка аварийной температуры. (Верхний блок лазеров)
         faultUpCam : Real := 45.0;   // Уставка аварийной температуры. (Верхний блок камер)
         faultDownLaser : Real := 45.0;   // Уставка аварийной температуры. (Нижний блок лазеров)
         faultDownCam : Real := 45.0;   // Уставка аварийной температуры. (Нижний блок камер)
         warnAir : Real := 50.0;   // Уставка предупреждающей температуры, для регулятора охладителя. (Воздух в пневмосистеме)
         warnUpLaser : Real := 32.0;   // Уставка предупреждающей температуры, для регулятора охладителя. (Верхний блок лазеров)
         warnUpCam : Real := 32.0;   // Уставка предупреждающей температуры, для регулятора охладителя. (Верхний блок камер)
         warnDownLaser : Real := 32.0;   // Уставка предупреждающей температуры, для регулятора охладителя. (Нижний блок лазеров)
         warnDownCam : Real := 32.0;   // Уставка предупреждающей температуры, для регулятора охладителя. (Нижний блок камер)
         reserv0 : Real;
      END_STRUCT;
      cleanTime : Struct   // Периодичность продувки
         tOnS : Real := 5.0;   // Время включения обдува, сек
         tOffMin : Real := 30.0;   // Время до следующего включения обдува, мин
      END_STRUCT;
      setPowerLasers : Struct   // Мощность лазеров. Или 0 - (откл.); или 100 - (вкл.)
         writeAll : Real := 100.0;   // Запись всех значений сразу
         upBlue1 : Real := 100.0;   // Активация верхнего синего лазера 1: *______________
         upBlue2 : Real := 100.0;   // Активация верхнего синего лазера 2: _*_____________
         upBlue3 : Real := 100.0;   // Активация верхнего синего лазера 3: __*____________
         upGreen1 : Real := 100.0;   // Активация верхнего зеленого лазера 1: ___*___________
         upGreen2 : Real := 100.0;   // Активация верхнего зеленого лазера 2: ____*__________
         upGreen3 : Real := 100.0;   // Активация верхнего зеленого лазера 3: _____*_________
         upBlue4 : Real := 100.0;   // Активация верхнего синего лазера 4: ______*________
         upBlue5 : Real := 100.0;   // Активация верхнего синего лазера 5: _______*_______
         upBlue6 : Real := 100.0;   // Активация верхнего синего лазера 6: ________*______
         upGreen4 : Real := 100.0;   // Активация верхнего зеленого лазера 4: _________*_____
         upGreen5 : Real := 100.0;   // Активация верхнего зеленого лазера 5: __________*____
         upGreen6 : Real := 100.0;   // Активация верхнего зеленого лазера 6: ___________*___
         upBlue7 : Real := 100.0;   // Активация верхнего синего лазера 7: ____________*__
         upBlue8 : Real := 100.0;   // Активация верхнего синего лазера 8: _____________*_
         upBlue9 : Real := 100.0;   // Активация верхнего синего лазера 9: ______________*
         downGreen1 : Real := 100.0;   // Активация нижнего зеленого лазера 1: *______________
         downGreen2 : Real := 100.0;   // Активация нижнего зеленого лазера 2: _*_____________
         downGreen3 : Real := 100.0;   // Активация нижнего зеленого лазера 3: __*____________
         downBlue1 : Real := 100.0;   // Активация нижнего синего лазера 1: ___*___________
         downBlue2 : Real := 100.0;   // Активация нижнего синего лазера 2: ____*__________
         downBlue3 : Real := 100.0;   // Активация нижнего синего лазера 3: _____*_________
         downGreen4 : Real := 100.0;   // Активация нижнего зеленого лазера 4: ______*________
         downGreen5 : Real := 100.0;   // Активация нижнего зеленого лазера 5: _______*_______
         downGreen6 : Real := 100.0;   // Активация нижнего зеленого лазера 6: ________*______
         downBlue4 : Real := 100.0;   // Активация нижнего синего лазера 4: _________*_____
         downBlue5 : Real := 100.0;   // Активация нижнего синего лазера 5: __________*____
         downBlue6 : Real := 100.0;   // Активация нижнего синего лазера 6: ___________*___
         downGreen7 : Real := 100.0;   // Активация нижнего зеленого лазера 7: ____________*__
         downGreen8 : Real := 100.0;   // Активация нижнего зеленого лазера 8: _____________*_
         downGreen9 : Real := 100.0;   // Активация нижнего зеленого лазера 9: ______________*
      END_STRUCT;
   END_VAR
BEGIN
END_DATA_BLOCK

// folder: Data_blocks

DATA_BLOCK "Initializing&Cooling_DB"   // DB1
{ S7_Optimized_Access := 'TRUE' }
VERSION : 0.1
// stored: InstanceOfName Initializing&Cooling
"Initializing&Cooling"
BEGIN
END_DATA_BLOCK

DATA_BLOCK "Blink_DB"   // DB2
{ S7_Optimized_Access := 'TRUE' }
VERSION : 0.1
// stored: InstanceOfName Blink
"Blink"
BEGIN
END_DATA_BLOCK

DATA_BLOCK "Inputs_Handler_DB"   // DB5
{ S7_Optimized_Access := 'TRUE' }
VERSION : 0.1
// stored: InstanceOfName Inputs_Handler
"Inputs_Handler"
BEGIN
END_DATA_BLOCK

DATA_BLOCK "Main_Block_db"   // DB6
{ S7_Optimized_Access := 'TRUE' }
VERSION : 0.1
// stored: InstanceOfName Main_Block
"Main_Block"
BEGIN
END_DATA_BLOCK

DATA_BLOCK "Laser&Synchro_db"   // DB7
{ S7_Optimized_Access := 'TRUE' }
VERSION : 0.1
// stored: InstanceOfName Laser&Synchro
"Laser&Synchro"
BEGIN
END_DATA_BLOCK

DATA_BLOCK "Outputs_Handler_DB"   // DB11
{ S7_Optimized_Access := 'TRUE' }
VERSION : 0.1
// stored: InstanceOfName Outputs_Handler
"Outputs_Handler"
BEGIN
END_DATA_BLOCK

// folder: Modbus

DATA_BLOCK "MB_DATA"   // DB10
{ S7_Optimized_Access := 'FALSE' }
VERSION : 0.1
   VAR
      s0 : Struct
         dw0 : Struct
            b0 : Bool;
            b1 : Bool := false;
            b2 : Bool := false;
            b3 : Bool := false;
            b4 : Bool := false;
            b5 : Bool := false;
            b6 : Bool := false;
            b7 : Bool := false;
            b8 : Bool := false;
            b9 : Bool := false;
            b10 : Bool := false;
            b11 : Bool := false;
            b12 : Bool := false;
            b13 : Bool := false;
            b14 : Bool := false;
            b15 : Bool := false;
         END_STRUCT;
         dw1 : Struct
            b0 : Bool;
            b1 : Bool := false;
            b2 : Bool := false;
            b3 : Bool := false;
            b4 : Bool := false;
            b5 : Bool := false;
            b6 : Bool := false;
            b7 : Bool := false;
            b8 : Bool := false;
            b9 : Bool := false;
            b10 : Bool := false;
            b11 : Bool := false;
            b12 : Bool := false;
            b13 : Bool := false;
            b14 : Bool := false;
            b15 : Bool := false;
         END_STRUCT;
         "dw2&3" : DWord;
         "dw4&5" : DWord := 16#0;
         "dw6&7" : DWord := 16#0;
         "dw8&9" : DWord := 16#0;
         "dw10&11" : DWord := 16#0;
         "dw12&13" : DWord := 16#0;
         dw14 : Word := 0;
         dw15 : Word := 0;
         dw16 : Word := 0;
         dw17 : Word := 0;
      END_STRUCT;
      dataAddr : DInt := 30001;
      len : Int := 18;
      disConn : Bool;
      conn : TCON_IP_v4;
   END_VAR
BEGIN
   conn.InterfaceId := 72;
   conn.ID := 1;
   conn.ActiveEstablished := true;
   conn.RemoteAddress.ADDR[1] := 10;
   conn.RemoteAddress.ADDR[2] := 97;
   conn.RemoteAddress.ADDR[3] := 189;
   conn.RemoteAddress.ADDR[4] := 33;
   conn.RemotePort := 502;
   conn.LocalPort := 0;
END_DATA_BLOCK

DATA_BLOCK "Modbus_Client_DB"   // DB16
{ S7_Optimized_Access := 'TRUE' }
VERSION : 0.1
// stored: InstanceOfName Modbus_Client
"Modbus_Client"
BEGIN
END_DATA_BLOCK

// folder: Socket_Send

DATA_BLOCK "Send_Connect"   // DB12
{ S7_Optimized_Access := 'TRUE' }
AUTHOR : SIMATIC
FAMILY : MC7Plus
NAME : TC_IP_v4
VERSION : 1.0
// stored: InstanceOfName TCON_IP_v4
"TCON_IP_v4"
BEGIN
   ID := 4;
   InterfaceId := 72;
   LocalPort := 2000;
END_DATA_BLOCK

DATA_BLOCK "Sock_RD_DB"   // DB14
{ S7_Optimized_Access := 'TRUE' }
VERSION : 0.1
// stored: InstanceOfName Sock_RD
"Sock_RD"
BEGIN
END_DATA_BLOCK

// folder: Socket_Write

DATA_BLOCK "WriteBuffer"   // DB8
{ S7_Optimized_Access := 'FALSE' }
VERSION : 0.1
   VAR
      resetErrorTrigg : Bool;   // Сброс аварии
      coolAirEn : Bool;
      setLasersManual : Struct   // Для ручного режима
         upBlueLasers123 : Bool := false;
         upGreenLasers123 : Bool := false;
         upBlueLasers456 : Bool := false;
         upGreenLasers456 : Bool := false;
         upBlueLasers789 : Bool := false;
         downGreenLasers123 : Bool := false;
         downBlueLasers123 : Bool := false;
         downGreenLasers465 : Bool := false;
         downBlueLasers456 : Bool := false;
         downGreenLasers789 : Bool := false;
      END_STRUCT;
      simulate : Struct   // Симуляция каналов. (для АО применимо из setPowerLasers)
         DI : Struct
            DI0 : USInt := 16#0;
            DI1 : USInt := 16#0;
            DI2 : USInt := 16#0;
            DI3 : USInt := 16#0;
            DI4 : USInt := 16#0;
            DI5 : USInt := 16#0;
            DI6 : USInt := 16#0;
            DI7 : USInt := 16#0;
            DI8 : USInt := 16#0;
            DI9 : USInt := 16#0;
            DI10 : USInt := 16#0;
            DI11 : USInt := 16#0;
            DI12 : USInt := 16#0;
            DI13 : USInt := 16#0;
            DI14 : USInt := 16#0;
            DI15 : USInt := 16#0;
         END_STRUCT;
         "DO" : Struct
            DO0 : USInt := 0;
            DO1 : USInt := 0;
            DO2 : USInt := 0;
            DO3 : USInt := 0;
            DO4 : USInt := 0;
            DO5 : USInt := 0;
            DO6 : USInt := 0;
            DO7 : USInt := 0;
            DO8 : USInt := 0;
            DO9 : USInt := 0;
            DO10 : USInt := 0;
            DO11 : USInt := 0;
            DO12 : USInt := 0;
            DO13 : USInt := 0;
            DO14 : USInt := 0;
            DO15 : USInt := 0;
            DO16 : USInt := 0;
            DO17 : USInt := 0;
            DO18 : USInt := 0;
            DO19 : USInt := 0;
            DO20 : USInt := 0;
            DO21 : USInt := 0;
            DO22 : USInt := 0;
            DO23 : USInt := 0;
            DO24 : USInt := 0;
            DO25 : USInt := 0;
            DO26 : USInt := 0;
            DO27 : USInt := 0;
            DO28 : USInt := 0;
            DO29 : USInt := 0;
            DO30 : USInt := 0;
            DO31 : USInt := 0;
         END_STRUCT;
         AI : Struct   // 0.0 -- симуляция отключена; от 0.0 до 0.001 -- запись 0.0; выше 0.001 -- запись любого числа.
            upTempLaser1 : Real := 0.0;
            upTempLaser2 : Real := 0.0;
            upTempCam1 : Real := 0.0;
            upTempCam2 : Real := 0.0;
            downTempLaser1 : Real := 0.0;
            downTempLaser2 : Real := 0.0;
            downTempCam1 : Real := 0.0;
            downTempCam2 : Real := 0.0;
            airTemperatur : Real := 0.0;
            reserv : Real := 0.0;
         END_STRUCT;
      END_STRUCT;
      setTemperatures : Struct   // Уставки температур
         faultUpLaser : Real := 0.0;
         faultUpCam : Real := 0.0;
         faultDownLaser : Real := 0.0;
         faultDownCam : Real := 0.0;
         warnAir : Real := 0.0;
         warnUpLaser : Real := 0.0;
         warnUpCam : Real := 0.0;
         warnDownLaser : Real := 0.0;
         warnDownCam : Real := 0.0;
         reserv0 : Real := 0.0;
      END_STRUCT;
      cleanTime : Struct   // Периодичность продувки
         tOnS : Real := 0.0;
         tOffMin : Real := 0.0;
      END_STRUCT;
      setPowerLasers : Struct   // Мощность лазеров (0 -- 100%)
         writeAll : Real := 0.0;
         upBlue1 : Real := 0.0;   // AO0.0
         upBlue2 : Real := 0.0;   // AO0.1
         upBlue3 : Real := 0.0;   // AO0.2
         upGreen1 : Real := 0.0;   // AO0.3
         upGreen2 : Real := 0.0;   // AO0.4
         upGreen3 : Real := 0.0;   // AO0.5
         upBlue4 : Real := 0.0;   // AO0.6
         upBlue5 : Real := 0.0;   // AO0.7
         upBlue6 : Real := 0.0;   // AO1.0
         upGreen4 : Real := 0.0;   // AO1.1
         upGreen5 : Real := 0.0;   // AO1.2
         upGreen6 : Real := 0.0;   // AO1.3
         upBlue7 : Real := 0.0;   // AO1.4
         upBlue8 : Real := 0.0;   // AO1.5
         upBlue9 : Real := 0.0;   // AO1.6
         downGreen1 : Real := 0.0;   // AO2.0
         downGreen2 : Real := 0.0;   // AO2.1
         downGreen3 : Real := 0.0;   // AO2.2
         downBlue1 : Real := 0.0;   // AO2.3
         downBlue2 : Real := 0.0;   // AO2.4
         downBlue3 : Real := 0.0;   // AO2.5
         downGreen4 : Real := 0.0;   // AO2.6
         downGreen5 : Real := 0.0;   // AO2.7
         downGreen6 : Real := 0.0;   // AO3.0
         downBlue4 : Real := 0.0;   // AO3.1
         downBlue5 : Real := 0.0;   // AO3.2
         downBlue6 : Real := 0.0;   // AO3.3
         downGreen7 : Real := 0.0;   // AO3.4
         downGreen8 : Real := 0.0;   // AO3.5
         downGreen9 : Real := 0.0;   // AO3.6
      END_STRUCT;
   END_VAR
BEGIN
END_DATA_BLOCK

DATA_BLOCK "Sock_WR_db"   // DB9
{ S7_Optimized_Access := 'TRUE' }
VERSION : 0.1
// stored: InstanceOfName Sock_WR
"Sock_WR"
BEGIN
END_DATA_BLOCK

DATA_BLOCK "TRCV_Connect"   // DB15
{ S7_Optimized_Access := 'TRUE' }
AUTHOR : SIMATIC
FAMILY : MC7Plus
NAME : TC_IP_v4
VERSION : 1.0
// stored: InstanceOfName TCON_IP_v4
"TCON_IP_v4"
BEGIN
   ID := 6;
   InterfaceId := 72;
   LocalPort := 2001;
END_DATA_BLOCK

// folder: (top level)

FUNCTION_BLOCK "Inputs_Handler"   // FB3, LAD
{ S7_Optimized_Access := 'TRUE' }
VERSION : 0.1
   VAR
      IEC_Timer_0_Instance : TON_TIME;
      ChangeReal_Instance : "ChangeReal";
   END_VAR
   VAR_TEMP
      reserv0 : Bool;
      reserv1 : Bool;
      reserv2 : Bool;
      AinMin : Bool;
      AinMax : Bool;
      valChanged : Bool;
   END_VAR
   VAR_TEMP   // added for the SCL form of the ladder/FBD networks
      _w1 : Bool;
   END_VAR
BEGIN

REGION Network 1: обработка входов
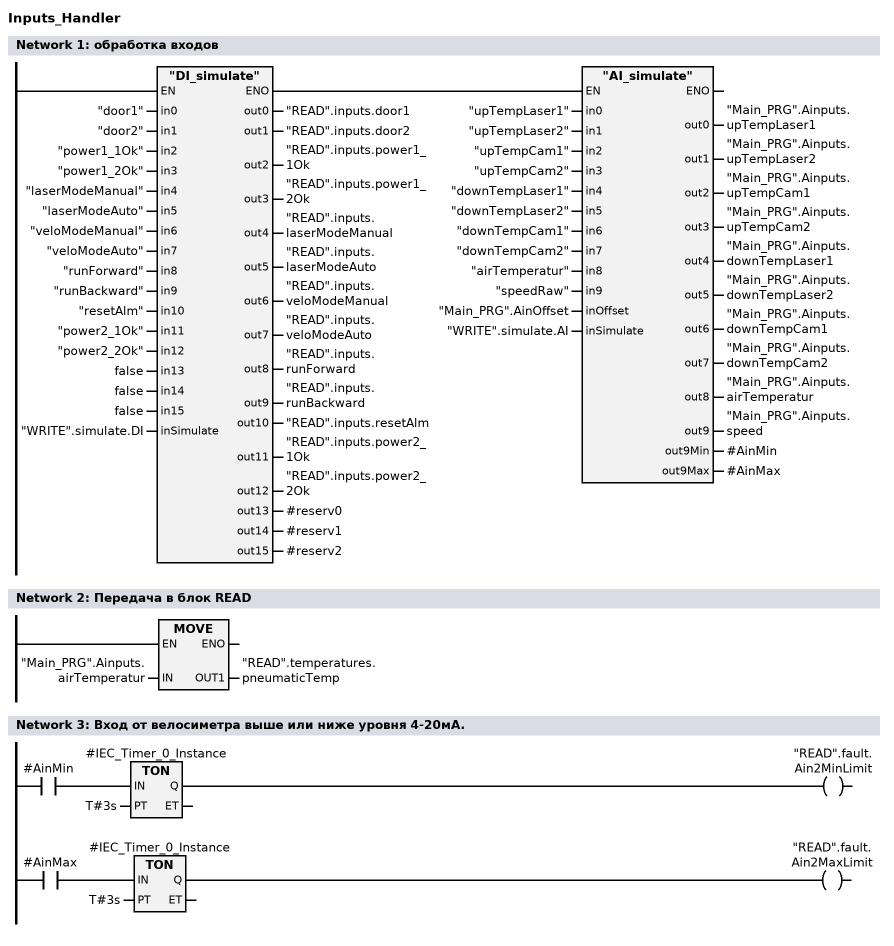
   RUNG wire#powerrail
      "DI_simulate"(in0 := "door1", in1 := "door2", in2 := "power1_1Ok", in3 := "power1_2Ok", in4 := "laserModeManual", in5 := "laserModeAuto", in6 := "veloModeManual", in7 := "veloModeAuto", in8 := "runForward", in9 := "runBackward", in10 := "resetAlm", in11 := "power2_1Ok", in12 := "power2_2Ok", in13 := false, in14 := false, in15 := false, inSimulate := "WRITE".simulate.DI, out0 => "READ".inputs.door1, out1 => "READ".inputs.door2, out2 => "READ".inputs.power1_1Ok, out3 => "READ".inputs.power1_2Ok, out4 => "READ".inputs.laserModeManual, out5 => "READ".inputs.laserModeAuto, out6 => "READ".inputs.veloModeManual, out7 => "READ".inputs.veloModeAuto, out8 => "READ".inputs.runForward, out9 => "READ".inputs.runBackward, out10 => "READ".inputs.resetAlm, out11 => "READ".inputs.power2_1Ok, out12 => "READ".inputs.power2_2Ok, out13 => #reserv0, out14 => #reserv1, out15 => #reserv2)
      "AI_simulate"(in0 := "upTempLaser1", in1 := "upTempLaser2", in2 := "upTempCam1", in3 := "upTempCam2", in4 := "downTempLaser1", in5 := "downTempLaser2", in6 := "downTempCam1", in7 := "downTempCam2", in8 := "airTemperatur", in9 := "speedRaw", inOffset := "Main_PRG".AinOffset, inSimulate := "WRITE".simulate.AI, out0 => "Main_PRG".Ainputs.upTempLaser1, out1 => "Main_PRG".Ainputs.upTempLaser2, out2 => "Main_PRG".Ainputs.upTempCam1, out3 => "Main_PRG".Ainputs.upTempCam2, out4 => "Main_PRG".Ainputs.downTempLaser1, out5 => "Main_PRG".Ainputs.downTempLaser2, out6 => "Main_PRG".Ainputs.downTempCam1, out7 => "Main_PRG".Ainputs.downTempCam2, out8 => "Main_PRG".Ainputs.airTemperatur, out9 => "Main_PRG".Ainputs.speed, out9Min => #AinMin, out9Max => #AinMax)
   END_RUNG
   // the same network as SCL:
   "DI_simulate"(in0 := "door1",
                 in1 := "door2",
                 in2 := "power1_1Ok",
                 in3 := "power1_2Ok",
                 in4 := "laserModeManual",
                 in5 := "laserModeAuto",
                 in6 := "veloModeManual",
                 in7 := "veloModeAuto",
                 in8 := "runForward",
                 in9 := "runBackward",
                 in10 := "resetAlm",
                 in11 := "power2_1Ok",
                 in12 := "power2_2Ok",
                 in13 := false,
                 in14 := false,
                 in15 := false,
                 inSimulate := "WRITE".simulate.DI,
                 out0 => "READ".inputs.door1,
                 out1 => "READ".inputs.door2,
                 out2 => "READ".inputs.power1_1Ok,
                 out3 => "READ".inputs.power1_2Ok,
                 out4 => "READ".inputs.laserModeManual,
                 out5 => "READ".inputs.laserModeAuto,
                 out6 => "READ".inputs.veloModeManual,
                 out7 => "READ".inputs.veloModeAuto,
                 out8 => "READ".inputs.runForward,
                 out9 => "READ".inputs.runBackward,
                 out10 => "READ".inputs.resetAlm,
                 out11 => "READ".inputs.power2_1Ok,
                 out12 => "READ".inputs.power2_2Ok,
                 out13 => #reserv0,
                 out14 => #reserv1,
                 out15 => #reserv2,
                 ENO => #_w1);
   IF #_w1 THEN
       "AI_simulate"(in0 := "upTempLaser1",
                     in1 := "upTempLaser2",
                     in2 := "upTempCam1",
                     in3 := "upTempCam2",
                     in4 := "downTempLaser1",
                     in5 := "downTempLaser2",
                     in6 := "downTempCam1",
                     in7 := "downTempCam2",
                     in8 := "airTemperatur",
                     in9 := "speedRaw",
                     inOffset := "Main_PRG".AinOffset,
                     inSimulate := "WRITE".simulate.AI,
                     out0 => "Main_PRG".Ainputs.upTempLaser1,
                     out1 => "Main_PRG".Ainputs.upTempLaser2,
                     out2 => "Main_PRG".Ainputs.upTempCam1,
                     out3 => "Main_PRG".Ainputs.upTempCam2,
                     out4 => "Main_PRG".Ainputs.downTempLaser1,
                     out5 => "Main_PRG".Ainputs.downTempLaser2,
                     out6 => "Main_PRG".Ainputs.downTempCam1,
                     out7 => "Main_PRG".Ainputs.downTempCam2,
                     out8 => "Main_PRG".Ainputs.airTemperatur,
                     out9 => "Main_PRG".Ainputs.speed,
                     out9Min => #AinMin,
                     out9Max => #AinMax);
   END_IF;
END_REGION

REGION Network 2: Передача в блок READ
   RUNG wire#powerrail
      Move(in := "Main_PRG".Ainputs.airTemperatur, out1 => "READ".temperatures.pneumaticTemp)
   END_RUNG
   // the same network as SCL:
   "READ".temperatures.pneumaticTemp := "Main_PRG".Ainputs.airTemperatur;
END_REGION

REGION Network 3: Вход от велосиметра выше или ниже уровня 4-20мА.
   #IEC_Timer_0_Instance(IN := #AinMin, PT := T#3s);   // TON
   "READ".fault.Ain2MinLimit := #IEC_Timer_0_Instance.Q;
   #IEC_Timer_0_Instance(IN := #AinMax, PT := T#3s);   // TON
   "READ".fault.Ain2MaxLimit := #IEC_Timer_0_Instance.Q;
END_REGION

REGION Network 4 (SCL): Переключает на другой вход, если он неисправен
   IF "Main_PRG".errUpTempLaser1 THEN
       "READ".temperatures.upLaserTemp := "Main_PRG".Ainputs.upTempLaser2;
   ELSE
       "READ".temperatures.upLaserTemp := "Main_PRG".Ainputs.upTempLaser1;
   END_IF;

   IF "Main_PRG".errUpTempCam1 THEN
       "READ".temperatures.upCamTemp := "Main_PRG".Ainputs.upTempCam2;
   ELSE
       "READ".temperatures.upCamTemp := "Main_PRG".Ainputs.upTempCam1;
   END_IF;

   IF "Main_PRG".errDownTempLaser1 THEN
       "READ".temperatures.downLaserTemp := "Main_PRG".Ainputs.downTempLaser2;
   ELSE
       "READ".temperatures.downLaserTemp := "Main_PRG".Ainputs.downTempLaser1;
   END_IF;

   IF "Main_PRG".errDownTempCam1 THEN
       "READ".temperatures.downCamTemp := "Main_PRG".Ainputs.downTempCam2;
   ELSE
       "READ".temperatures.downCamTemp := "Main_PRG".Ainputs.downTempCam1;
   END_IF;
END_REGION
END_FUNCTION_BLOCK

FUNCTION_BLOCK "Initializing&Cooling"   // FB7, LAD
{ S7_Optimized_Access := 'TRUE' }
VERSION : 0.1
   VAR_INPUT
      resetTrigg : Bool;
   END_VAR
   VAR_OUTPUT
      iniOk : Bool;
      initializing : Bool;
      faultTrigg : Bool;
      warning : Bool;
      toAirClean : Bool;
      toCoolUpLaser : Bool;
      toCoolUpCam : Bool;
      toCoolDownLaser : Bool;
      toCoolDownCam : Bool;
   END_VAR
   VAR
      IEC_Timer_0_Instance : TON_TIME;
      "4Hysteresis_Instance" : "4Hysteresis";
      "5Hysteresis_Instance" : "5Hysteresis";
      initializing_Instance : "initializing";
      interInitializing : Bool;
      iniErr : Bool;
      IEC_Timer_0_Instance_2 : TON_TIME;
      IEC_Timer_0_Instance_3 : TOF_TIME;
      fault : Bool;
      positiv0 : Bool;
      IEC_Timer_0_Instance_4 : TOF_TIME;
      IEC_Timer_0_Instance_1 : TON_TIME;
      IEC_Timer_0_Instance_5 : TON_TIME;
      IEC_Timer_0_Instance_6 : TON_TIME;
      IEC_Timer_0_Instance_7 : TON_TIME;
      IEC_Timer_0_Instance_8 : TON_TIME;
      IEC_Timer_0_Instance_9 : TON_TIME;
   END_VAR
   VAR_TEMP
      anyFault : Bool;
      interAirOn : Bool;
      interWarnPneum : Bool;
      rstErrTrigg : Bool;
   END_VAR
   VAR_TEMP   // added for the SCL form of the ladder/FBD networks
      _w1 : Bool;
   END_VAR
BEGIN

REGION Network 1: Сброс триггера аварий
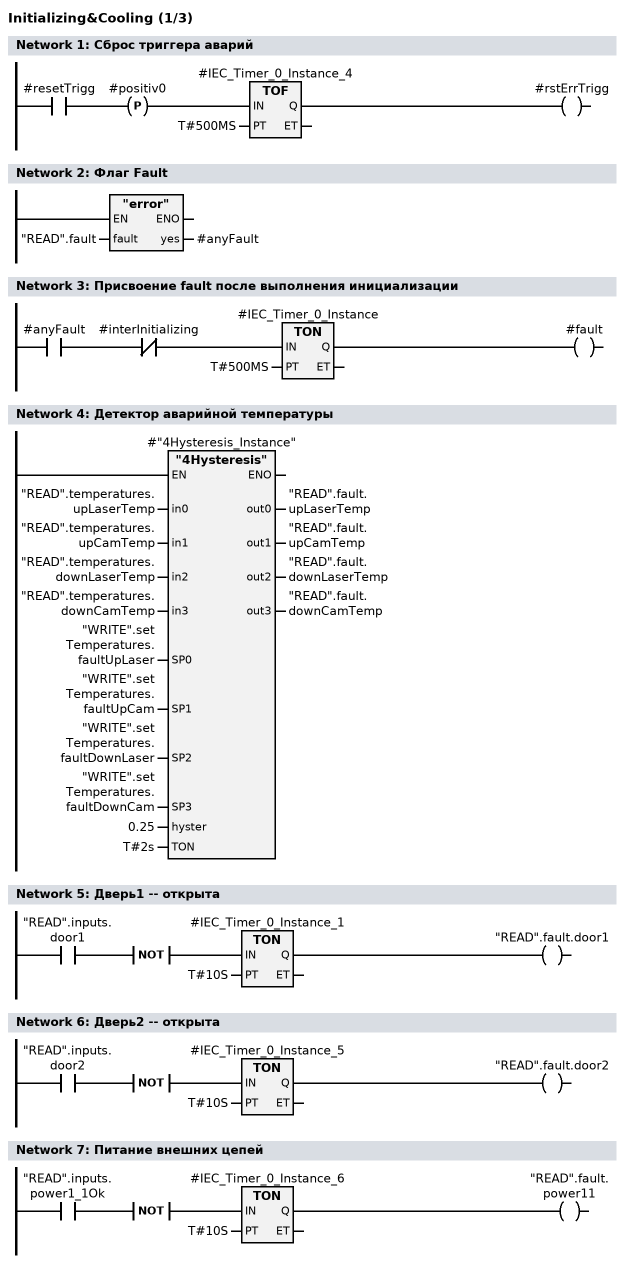
   #_w1 := #resetTrigg AND NOT #positiv0;   // rising edge
   #positiv0 := #resetTrigg;
   #IEC_Timer_0_Instance_4(IN := #_w1, PT := T#500MS);   // TOF
   #rstErrTrigg := #IEC_Timer_0_Instance_4.Q;
END_REGION

REGION Network 2: Флаг Fault
   RUNG wire#powerrail
      "error"(fault := "READ".fault, yes => #anyFault)
   END_RUNG
   // the same network as SCL:
   "error"(fault := "READ".fault, yes => #anyFault);
END_REGION

REGION Network 3: Присвоение fault после выполнения инициализации
   #IEC_Timer_0_Instance(IN := #anyFault AND NOT #interInitializing, PT := T#500MS);   // TON
   #fault := #IEC_Timer_0_Instance.Q;
END_REGION

REGION Network 4: Детектор аварийной температуры
   RUNG wire#powerrail
      #"4Hysteresis_Instance"(in0 := "READ".temperatures.upLaserTemp, in1 := "READ".temperatures.upCamTemp, in2 := "READ".temperatures.downLaserTemp, in3 := "READ".temperatures.downCamTemp, SP0 := "WRITE".setTemperatures.faultUpLaser, SP1 := "WRITE".setTemperatures.faultUpCam, SP2 := "WRITE".setTemperatures.faultDownLaser, SP3 := "WRITE".setTemperatures.faultDownCam, hyster := 0.25, TON := T#2s, out0 => "READ".fault.upLaserTemp, out1 => "READ".fault.upCamTemp, out2 => "READ".fault.downLaserTemp, out3 => "READ".fault.downCamTemp)
   END_RUNG
   // the same network as SCL:
   #"4Hysteresis_Instance"(in0 := "READ".temperatures.upLaserTemp,   // "4Hysteresis"
                           in1 := "READ".temperatures.upCamTemp,
                           in2 := "READ".temperatures.downLaserTemp,
                           in3 := "READ".temperatures.downCamTemp,
                           SP0 := "WRITE".setTemperatures.faultUpLaser,
                           SP1 := "WRITE".setTemperatures.faultUpCam,
                           SP2 := "WRITE".setTemperatures.faultDownLaser,
                           SP3 := "WRITE".setTemperatures.faultDownCam,
                           hyster := 0.25,
                           TON := T#2s,
                           out0 => "READ".fault.upLaserTemp,
                           out1 => "READ".fault.upCamTemp,
                           out2 => "READ".fault.downLaserTemp,
                           out3 => "READ".fault.downCamTemp);
END_REGION

REGION Network 5: Дверь1 -- открыта
   #IEC_Timer_0_Instance_1(IN := NOT "READ".inputs.door1, PT := T#10S);   // TON
   "READ".fault.door1 := #IEC_Timer_0_Instance_1.Q;
END_REGION

REGION Network 6: Дверь2 -- открыта
   #IEC_Timer_0_Instance_5(IN := NOT "READ".inputs.door2, PT := T#10S);   // TON
   "READ".fault.door2 := #IEC_Timer_0_Instance_5.Q;
END_REGION

REGION Network 7: Питание внешних цепей
   #IEC_Timer_0_Instance_6(IN := NOT "READ".inputs.power1_1Ok, PT := T#10S);   // TON
   "READ".fault.power11 := #IEC_Timer_0_Instance_6.Q;
END_REGION

REGION Network 8: Питание внутренних цепей
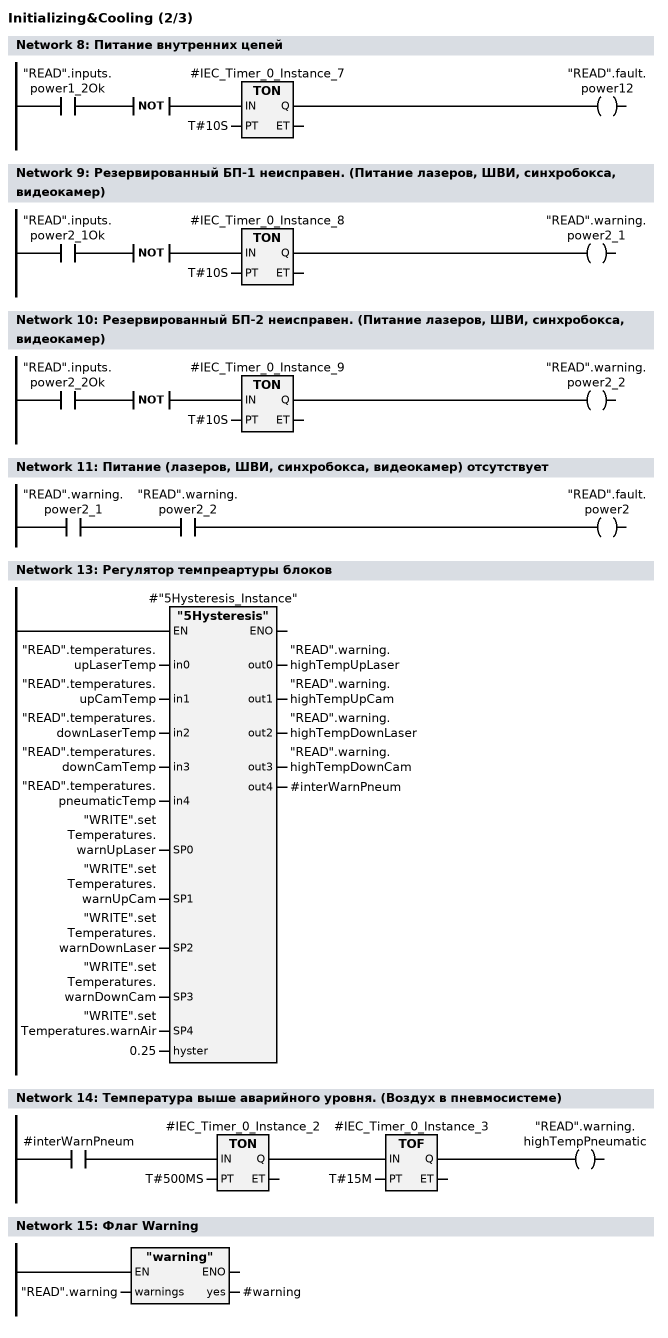
   #IEC_Timer_0_Instance_7(IN := NOT "READ".inputs.power1_2Ok, PT := T#10S);   // TON
   "READ".fault.power12 := #IEC_Timer_0_Instance_7.Q;
END_REGION

REGION Network 9: Резервированный БП-1 неисправен. (Питание лазеров, ШВИ, синхробокса, видеокамер)
   #IEC_Timer_0_Instance_8(IN := NOT "READ".inputs.power2_1Ok, PT := T#10S);   // TON
   "READ".warning.power2_1 := #IEC_Timer_0_Instance_8.Q;
END_REGION

REGION Network 10: Резервированный БП-2 неисправен. (Питание лазеров, ШВИ, синхробокса, видеокамер)
   #IEC_Timer_0_Instance_9(IN := NOT "READ".inputs.power2_2Ok, PT := T#10S);   // TON
   "READ".warning.power2_2 := #IEC_Timer_0_Instance_9.Q;
END_REGION

REGION Network 11: Питание (лазеров, ШВИ, синхробокса, видеокамер) отсутствует
   RUNG wire#powerrail
      Contact( "READ".warning.power2_1 )
      Contact( "READ".warning.power2_2 )
      Coil( "READ".fault.power2 )
   END_RUNG
   // the same network as SCL:
   "READ".fault.power2 := "READ".warning.power2_1 AND "READ".warning.power2_2;
END_REGION

REGION Network 12 (SCL): вывод аварии, если оба канала температур в блоке лазеров/камер неисправны
   "READ".fault.upLaserAllCh := "Main_PRG".errUpTempLaser1 AND "Main_PRG".errUpTempLaser2;
   "READ".fault.upCamAllCh := "Main_PRG".errUpTempCam1 AND "Main_PRG".errUpTempCam2;
   "READ".fault.downLaserAllCh := "Main_PRG".errDownTempLaser1 AND "Main_PRG".errDownTempLaser2;
   "READ".fault.downCamAllCh := "Main_PRG".errDownTempCam1 AND "Main_PRG".errDownTempCam2;
END_REGION

REGION Network 13: Регулятор темпреартуры блоков
   RUNG wire#powerrail
      #"5Hysteresis_Instance"(in0 := "READ".temperatures.upLaserTemp, in1 := "READ".temperatures.upCamTemp, in2 := "READ".temperatures.downLaserTemp, in3 := "READ".temperatures.downCamTemp, in4 := "READ".temperatures.pneumaticTemp, SP0 := "WRITE".setTemperatures.warnUpLaser, SP1 := "WRITE".setTemperatures.warnUpCam, SP2 := "WRITE".setTemperatures.warnDownLaser, SP3 := "WRITE".setTemperatures.warnDownCam, SP4 := "WRITE".setTemperatures.warnAir, hyster := 0.25, out0 => "READ".warning.highTempUpLaser, out1 => "READ".warning.highTempUpCam, out2 => "READ".warning.highTempDownLaser, out3 => "READ".warning.highTempDownCam, out4 => #interWarnPneum)
   END_RUNG
   // the same network as SCL:
   #"5Hysteresis_Instance"(in0 := "READ".temperatures.upLaserTemp,   // "5Hysteresis"
                           in1 := "READ".temperatures.upCamTemp,
                           in2 := "READ".temperatures.downLaserTemp,
                           in3 := "READ".temperatures.downCamTemp,
                           in4 := "READ".temperatures.pneumaticTemp,
                           SP0 := "WRITE".setTemperatures.warnUpLaser,
                           SP1 := "WRITE".setTemperatures.warnUpCam,
                           SP2 := "WRITE".setTemperatures.warnDownLaser,
                           SP3 := "WRITE".setTemperatures.warnDownCam,
                           SP4 := "WRITE".setTemperatures.warnAir,
                           hyster := 0.25,
                           out0 => "READ".warning.highTempUpLaser,
                           out1 => "READ".warning.highTempUpCam,
                           out2 => "READ".warning.highTempDownLaser,
                           out3 => "READ".warning.highTempDownCam,
                           out4 => #interWarnPneum);
END_REGION

REGION Network 14: Температура выше аварийного уровня. (Воздух в пневмосистеме)
   #IEC_Timer_0_Instance_2(IN := #interWarnPneum, PT := T#500MS);   // TON
   #IEC_Timer_0_Instance_3(IN := #IEC_Timer_0_Instance_2.Q, PT := T#15M);   // TOF
   "READ".warning.highTempPneumatic := #IEC_Timer_0_Instance_3.Q;
END_REGION

REGION Network 15: Флаг Warning
   RUNG wire#powerrail
      "warning"(warnings := "READ".warning, yes => #warning)
   END_RUNG
   // the same network as SCL:
   "warning"(warnings := "READ".warning, yes => #warning);
END_REGION

REGION Network 16: Продувка и охлаждение при первом включении
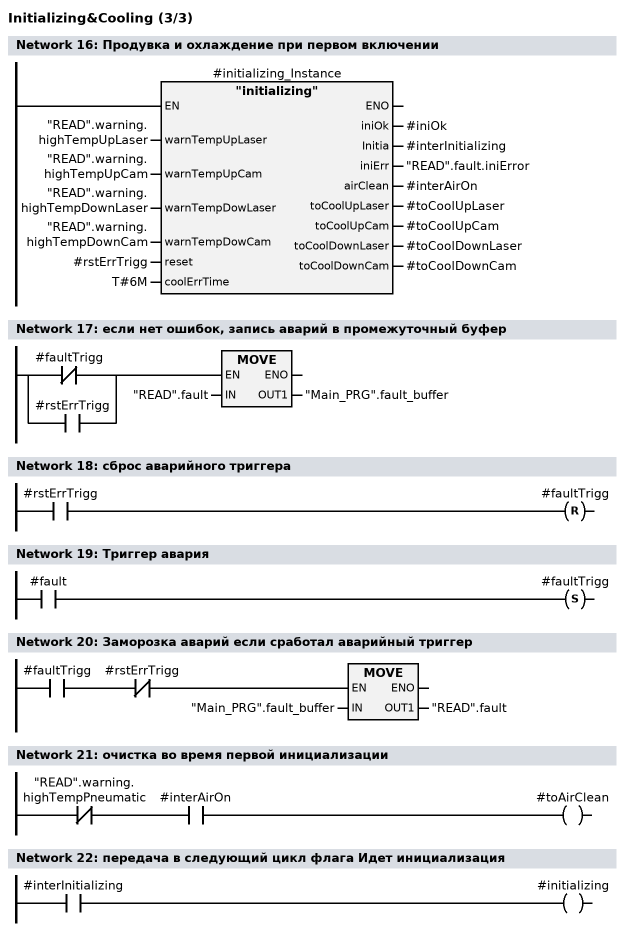
   RUNG wire#powerrail
      #initializing_Instance(warnTempUpLaser := "READ".warning.highTempUpLaser, warnTempUpCam := "READ".warning.highTempUpCam, warnTempDowLaser := "READ".warning.highTempDownLaser, warnTempDowCam := "READ".warning.highTempDownCam, reset := #rstErrTrigg, coolErrTime := T#6M, iniOk => #iniOk, Initia => #interInitializing, iniErr => "READ".fault.iniError, airClean => #interAirOn, toCoolUpLaser => #toCoolUpLaser, toCoolUpCam => #toCoolUpCam, toCoolDownLaser => #toCoolDownLaser, toCoolDownCam => #toCoolDownCam)
   END_RUNG
   // the same network as SCL:
   #initializing_Instance(warnTempUpLaser := "READ".warning.highTempUpLaser,   // "initializing"
                          warnTempUpCam := "READ".warning.highTempUpCam,
                          warnTempDowLaser := "READ".warning.highTempDownLaser,
                          warnTempDowCam := "READ".warning.highTempDownCam,
                          reset := #rstErrTrigg,
                          coolErrTime := T#6M,
                          iniOk => #iniOk,
                          Initia => #interInitializing,
                          iniErr => "READ".fault.iniError,
                          airClean => #interAirOn,
                          toCoolUpLaser => #toCoolUpLaser,
                          toCoolUpCam => #toCoolUpCam,
                          toCoolDownLaser => #toCoolDownLaser,
                          toCoolDownCam => #toCoolDownCam);
END_REGION

REGION Network 17: если нет ошибок, запись аварий в промежуточный буфер
   RUNG wire#powerrail
      I_Contact( #faultTrigg )
      wire#w1
      Move(in := "READ".fault, out1 => "Main_PRG".fault_buffer)
   END_RUNG
   RUNG wire#powerrail
      Contact( #rstErrTrigg )
   END_RUNG wire#w1
   // the same network as SCL:
   IF NOT #faultTrigg OR #rstErrTrigg THEN "Main_PRG".fault_buffer := "READ".fault; END_IF;
END_REGION

REGION Network 18: сброс аварийного триггера
   RUNG wire#powerrail
      Contact( #rstErrTrigg )
      R_Coil( #faultTrigg )
   END_RUNG
   // the same network as SCL:
   IF #rstErrTrigg THEN #faultTrigg := FALSE; END_IF;
END_REGION

REGION Network 19: Триггер авария
   RUNG wire#powerrail
      Contact( #fault )
      S_Coil( #faultTrigg )
   END_RUNG
   // the same network as SCL:
   IF #fault THEN #faultTrigg := TRUE; END_IF;
END_REGION

REGION Network 20: Заморозка аварий если сработал аварийный триггер
   RUNG wire#powerrail
      Contact( #faultTrigg )
      I_Contact( #rstErrTrigg )
      Move(in := "Main_PRG".fault_buffer, out1 => "READ".fault)
   END_RUNG
   // the same network as SCL:
   IF #faultTrigg AND NOT #rstErrTrigg THEN "READ".fault := "Main_PRG".fault_buffer; END_IF;
END_REGION

REGION Network 21: очистка во время первой инициализации
   RUNG wire#powerrail
      I_Contact( "READ".warning.highTempPneumatic )
      Contact( #interAirOn )
      Coil( #toAirClean )
   END_RUNG
   // the same network as SCL:
   #toAirClean := NOT "READ".warning.highTempPneumatic AND #interAirOn;
END_REGION

REGION Network 22: передача в следующий цикл флага Идет инициализация
   RUNG wire#powerrail
      Contact( #interInitializing )
      Coil( #initializing )
   END_RUNG
   // the same network as SCL:
   #initializing := #interInitializing;
END_REGION
END_FUNCTION_BLOCK

FUNCTION_BLOCK "Main_Block"   // FB9, LAD
{ S7_Optimized_Access := 'TRUE' }
VERSION : 0.1
   VAR_INPUT
      faultTrigg : Bool;
      warning : Bool;
      initializing : Bool;
      initOk : Bool;
      outEnable : Bool;
      velocimeterModeManual : Bool;
      velocimeterModeAuto : Bool;
      revers : Bool;
      synchroOn : Bool;
      airTon : Real;
      airToff : Real;
      speed : Real;
   END_VAR
   VAR_OUTPUT
      RUN : Bool;
      airOn : Bool;
      veloLaser_En : Bool;
      veloShut_En : Bool;
      coolUpLaserOn : Bool;
      coolUpCamOn : Bool;
      coolDownLaserOn : Bool;
      coolDownCamOn : Bool;
      redLamp : Bool;
      greenLamp : Bool;
      dirForward : Bool;
      dirBackward : Bool;
      greenLampStat : Bool;
      redLampStat : Bool;
   END_VAR
   VAR
      interPneum : Bool;
      CTUout : Bool;
      P_TRIG_0 : Bool;
      IEC_Timer_0_Instance : TON_TIME;
      IEC_Timer_0_Instance_1 : TON_TIME;
      Blink_Instance : "Blink";
   END_VAR
   VAR RETAIN
      IEC_Counter_0_Instance : CTU_INT;
   END_VAR
   VAR
      Blink_Instance_1 : "Blink";
      P_TRIG_1 : Bool;
      BlinkRUN : Bool;
      IEC_Timer_0_Instance_2 : TON_TIME;
      IEC_Timer_0_Instance_3 : TON_TIME;
      IEC_Timer_0_Instance_4 : TOF_TIME;
   END_VAR
   VAR_TEMP
      pneumaticEn : Bool;
      interPneumDelay : Bool;
      inter0AirTon : Real;
      inter0AirToff : Real;
      interAirTon : DInt;
      interAirToff : DInt;
      blinkLamp : Bool;
   END_VAR
   VAR_TEMP   // added for the SCL form of the ladder/FBD networks
      _w1 : Bool;
      _w2 : Bool;
   END_VAR
BEGIN

REGION Network 1 (SCL): Пересчет в минуты и секунды для констант таймера продувки
   #inter0AirTon := #airTon * 1000;
   #interAirTon := REAL_TO_DINT(#inter0AirTon);

   #inter0AirToff := #airToff * 60000;
   #interAirToff := REAL_TO_DINT(#inter0AirToff);
END_REGION

REGION Network 2: Если нет аварий, инициал-Ок, скорость >= 0, есть сигнал с цеха -- тогда Пуск
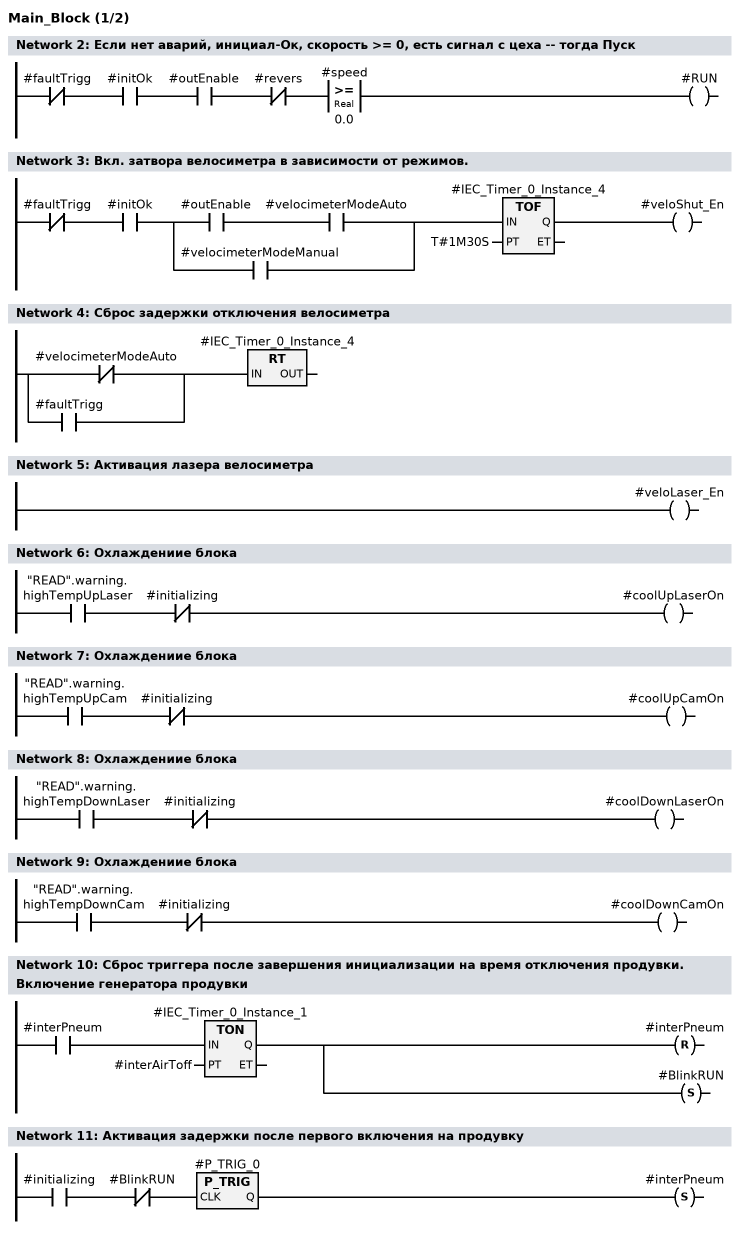
   RUNG wire#powerrail
      I_Contact( #faultTrigg )
      Contact( #initOk )
      Contact( #outEnable )
      I_Contact( #revers )
      { S7_Templates := "SrcType := Real" } GE_Contact(in1 := #speed, in2 := 0.0)
      Coil( #RUN )
   END_RUNG
   // the same network as SCL:
   #RUN := NOT #faultTrigg AND #initOk AND #outEnable AND NOT #revers AND (#speed >= 0.0);
END_REGION

REGION Network 3: Вкл. затвора велосиметра в зависимости от режимов.
   #IEC_Timer_0_Instance_4(IN := NOT #faultTrigg AND #initOk AND ((#outEnable AND #velocimeterModeAuto) OR #velocimeterModeManual),   // TOF
                           PT := T#1M30S);
   #veloShut_En := #IEC_Timer_0_Instance_4.Q;
END_REGION

REGION Network 4: Сброс задержки отключения велосиметра
   RUNG wire#powerrail
      I_Contact( #velocimeterModeAuto )
      wire#w1
      RT_Coil( #IEC_Timer_0_Instance_4 )
   END_RUNG
   RUNG wire#powerrail
      Contact( #faultTrigg )
   END_RUNG wire#w1
   // the same network as SCL:
   IF NOT #velocimeterModeAuto OR #faultTrigg THEN RESET_TIMER(#IEC_Timer_0_Instance_4); END_IF;
END_REGION

REGION Network 5: Активация лазера велосиметра
   RUNG wire#powerrail
      Coil( #veloLaser_En )
   END_RUNG
   // the same network as SCL:
   #veloLaser_En := TRUE;
END_REGION

REGION Network 6: Охлаждениие блока
   RUNG wire#powerrail
      Contact( "READ".warning.highTempUpLaser )
      I_Contact( #initializing )
      Coil( #coolUpLaserOn )
   END_RUNG
   // the same network as SCL:
   #coolUpLaserOn := "READ".warning.highTempUpLaser AND NOT #initializing;
END_REGION

REGION Network 7: Охлаждениие блока
   RUNG wire#powerrail
      Contact( "READ".warning.highTempUpCam )
      I_Contact( #initializing )
      Coil( #coolUpCamOn )
   END_RUNG
   // the same network as SCL:
   #coolUpCamOn := "READ".warning.highTempUpCam AND NOT #initializing;
END_REGION

REGION Network 8: Охлаждениие блока
   RUNG wire#powerrail
      Contact( "READ".warning.highTempDownLaser )
      I_Contact( #initializing )
      Coil( #coolDownLaserOn )
   END_RUNG
   // the same network as SCL:
   #coolDownLaserOn := "READ".warning.highTempDownLaser AND NOT #initializing;
END_REGION

REGION Network 9: Охлаждениие блока
   RUNG wire#powerrail
      Contact( "READ".warning.highTempDownCam )
      I_Contact( #initializing )
      Coil( #coolDownCamOn )
   END_RUNG
   // the same network as SCL:
   #coolDownCamOn := "READ".warning.highTempDownCam AND NOT #initializing;
END_REGION

REGION Network 10: Сброс триггера после завершения инициализации на время отключения продувки. Включение генератора продувки
   #IEC_Timer_0_Instance_1(IN := #interPneum, PT := #interAirToff);   // TON
   IF #IEC_Timer_0_Instance_1.Q THEN
       #interPneum := FALSE;
       #BlinkRUN := TRUE;
   END_IF;
END_REGION

REGION Network 11: Активация задержки после первого включения на продувку
   RUNG wire#powerrail
      Contact( #initializing )
      I_Contact( #BlinkRUN )
      P_Trig( #P_TRIG_0 )
      S_Coil( #interPneum )
   END_RUNG
   // the same network as SCL:
   #_w1 := #initializing AND NOT #BlinkRUN;
   #_w2 := #_w1 AND NOT #P_TRIG_0;   // rising edge
   #P_TRIG_0 := #_w1;
   IF #_w2 THEN #interPneum := TRUE; END_IF;
END_REGION

REGION Network 12: генератор продувки
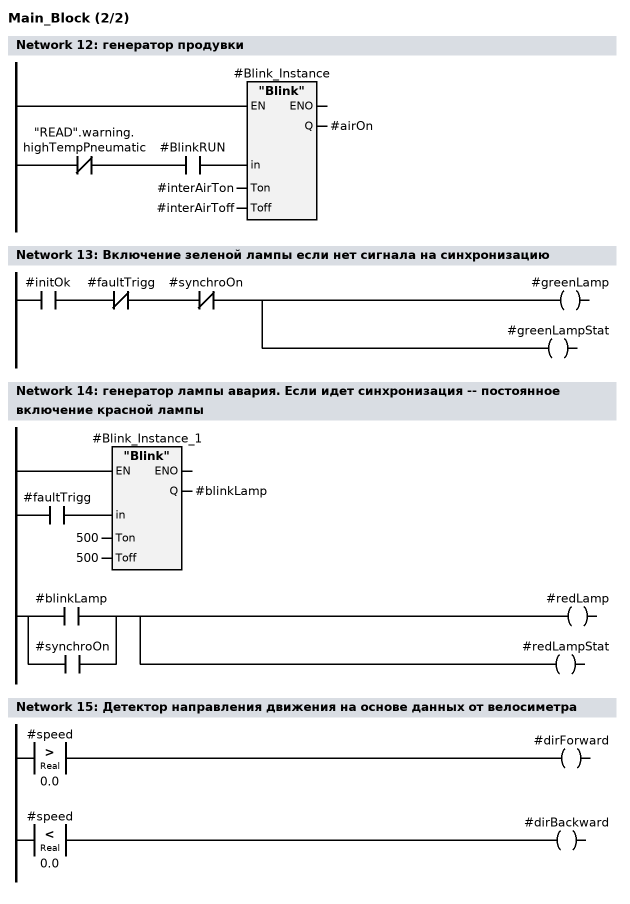
   RUNG wire#powerrail
      #Blink_Instance(in := wire#w1, Ton := #interAirTon, Toff := #interAirToff, Q => #airOn)
   END_RUNG
   RUNG wire#powerrail
      I_Contact( "READ".warning.highTempPneumatic )
      Contact( #BlinkRUN )
   END_RUNG wire#w1
   // the same network as SCL:
   #Blink_Instance(in := NOT "READ".warning.highTempPneumatic AND #BlinkRUN,   // "Blink"
                   Ton := #interAirTon,
                   Toff := #interAirToff,
                   Q => #airOn);
END_REGION

REGION Network 13: Включение зеленой лампы если нет сигнала на синхронизацию
   RUNG wire#powerrail
      Contact( #initOk )
      I_Contact( #faultTrigg )
      I_Contact( #synchroOn )
      wire#w1
      Coil( #greenLamp )
   END_RUNG
   RUNG wire#w1
      Coil( #greenLampStat )
   END_RUNG
   // the same network as SCL:
   #greenLamp := #initOk AND NOT #faultTrigg AND NOT #synchroOn;
   #greenLampStat := #greenLamp;
END_REGION

REGION Network 14: генератор лампы авария. Если идет синхронизация -- постоянное включение красной лампы
   RUNG wire#powerrail
      #Blink_Instance_1(in := wire#w1, Ton := 500, Toff := 500, Q => #blinkLamp)
   END_RUNG
   RUNG wire#powerrail
      Contact( #faultTrigg )
   END_RUNG wire#w1
   RUNG wire#powerrail
      Contact( #blinkLamp )
      wire#w2
      Coil( #redLamp )
   END_RUNG
   RUNG wire#powerrail
      Contact( #synchroOn )
   END_RUNG wire#w2
   RUNG wire#w2
      Coil( #redLampStat )
   END_RUNG
   // the same network as SCL:
   #Blink_Instance_1(in := #faultTrigg, Ton := 500, Toff := 500, Q => #blinkLamp);   // "Blink"
   #redLamp := #blinkLamp OR #synchroOn;
   #redLampStat := #redLamp;
END_REGION

REGION Network 15: Детектор направления движения на основе данных от велосиметра
   RUNG wire#powerrail
      { S7_Templates := "SrcType := Real" } GT_Contact(in1 := #speed, in2 := 0.0)
      Coil( #dirForward )
   END_RUNG
   RUNG wire#powerrail
      { S7_Templates := "SrcType := Real" } LT_Contact(in1 := #speed, in2 := 0.0)
      Coil( #dirBackward )
   END_RUNG
   // the same network as SCL:
   #dirForward := #speed > 0.0;
   #dirBackward := #speed < 0.0;
END_REGION
END_FUNCTION_BLOCK

FUNCTION_BLOCK "Laser&Synchro"   // FB11, LAD
{ S7_Optimized_Access := 'TRUE' }
VERSION : 0.1
   VAR_INPUT
      run : Bool;
      laserModeM : Bool;
      laserModeA : Bool;
      enBlueUpLaser123 : Bool;
      enGreenUpLaser123 : Bool;
      enBlueUpLaser456 : Bool;
      enGreenUpLaser456 : Bool;
      enBlueUpLaser789 : Bool;
      enGreenDownLaser123 : Bool;
      enBlueDownLaser123 : Bool;
      enGreenDownLaser456 : Bool;
      enBlueDownLaser456 : Bool;
      enGreenDownLaser789 : Bool;
      veloEN : Bool;
      iniOk : Bool;
      faultTrigg : Bool;
   END_VAR
   VAR_OUTPUT
      blueUpLaser_123 : Bool;
      greenUpLaser_123 : Bool;
      blueUpLaser_456 : Bool;
      greenUpLaser_456 : Bool;
      blueUpLaser_789 : Bool;
      greenDownLaser_123 : Bool;
      blueDownLaser_123 : Bool;
      greenDownLaser_456 : Bool;
      blueDownLaser_456 : Bool;
      greenDownLaser_789 : Bool;
      synchroOn : Bool;
      disSynchro : Bool;
   END_VAR
   VAR
      IEC_Timer_0_Instance : TOF_TIME;
   END_VAR
   VAR_TEMP
      lasersOn : Bool;
   END_VAR
BEGIN

REGION Network 1: Задержка отключения лазеров
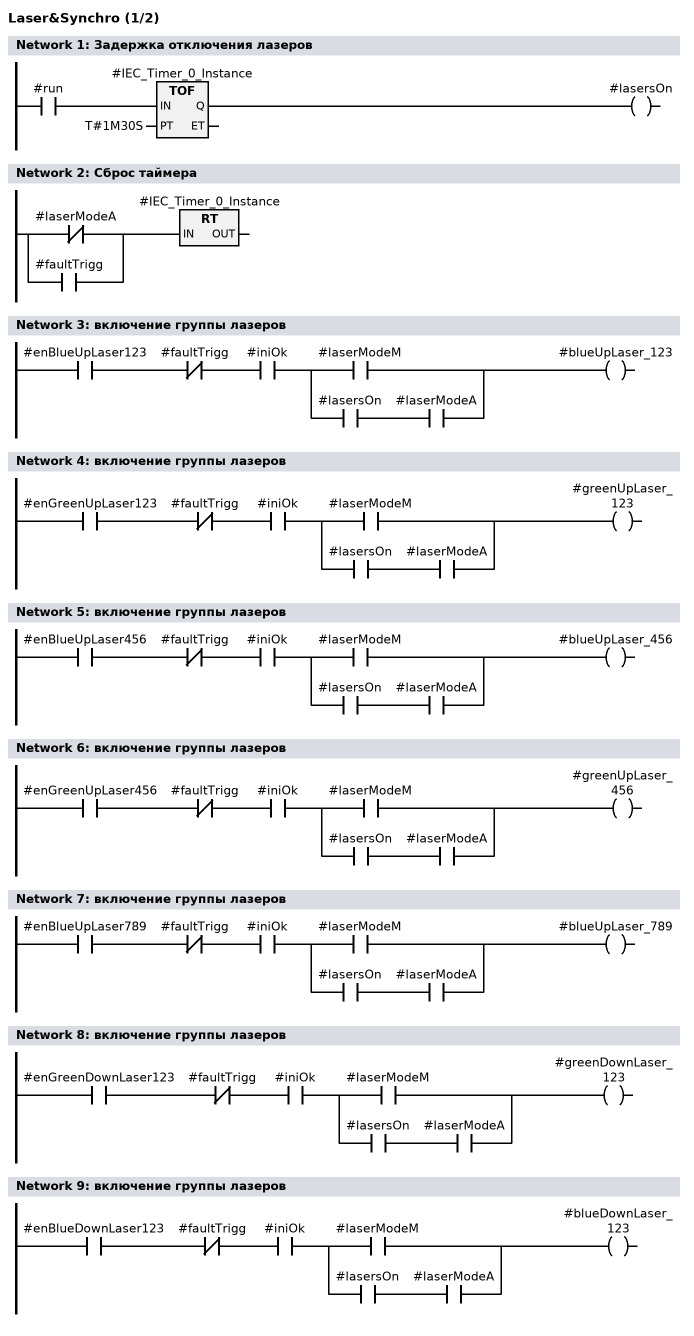
   #IEC_Timer_0_Instance(IN := #run, PT := T#1M30S);   // TOF
   #lasersOn := #IEC_Timer_0_Instance.Q;
END_REGION

REGION Network 2: Сброс таймера
   RUNG wire#powerrail
      I_Contact( #laserModeA )
      wire#w1
      RT_Coil( #IEC_Timer_0_Instance )
   END_RUNG
   RUNG wire#powerrail
      Contact( #faultTrigg )
   END_RUNG wire#w1
   // the same network as SCL:
   IF NOT #laserModeA OR #faultTrigg THEN RESET_TIMER(#IEC_Timer_0_Instance); END_IF;
END_REGION

REGION Network 3: включение группы лазеров
   RUNG wire#powerrail
      Contact( #enBlueUpLaser123 )
      I_Contact( #faultTrigg )
      Contact( #iniOk )
      wire#w1
      Contact( #laserModeM )
      wire#w2
      Coil( #blueUpLaser_123 )
   END_RUNG
   RUNG wire#w1
      Contact( #lasersOn )
      Contact( #laserModeA )
   END_RUNG wire#w2
   // the same network as SCL:
   #blueUpLaser_123 := #enBlueUpLaser123 AND NOT #faultTrigg AND #iniOk AND (#laserModeM OR (#lasersOn AND #laserModeA));
END_REGION

REGION Network 4: включение группы лазеров
   RUNG wire#powerrail
      Contact( #enGreenUpLaser123 )
      I_Contact( #faultTrigg )
      Contact( #iniOk )
      wire#w1
      Contact( #laserModeM )
      wire#w2
      Coil( #greenUpLaser_123 )
   END_RUNG
   RUNG wire#w1
      Contact( #lasersOn )
      Contact( #laserModeA )
   END_RUNG wire#w2
   // the same network as SCL:
   #greenUpLaser_123 := #enGreenUpLaser123 AND NOT #faultTrigg AND #iniOk AND (#laserModeM OR (#lasersOn AND #laserModeA));
END_REGION

REGION Network 5: включение группы лазеров
   RUNG wire#powerrail
      Contact( #enBlueUpLaser456 )
      I_Contact( #faultTrigg )
      Contact( #iniOk )
      wire#w1
      Contact( #laserModeM )
      wire#w2
      Coil( #blueUpLaser_456 )
   END_RUNG
   RUNG wire#w1
      Contact( #lasersOn )
      Contact( #laserModeA )
   END_RUNG wire#w2
   // the same network as SCL:
   #blueUpLaser_456 := #enBlueUpLaser456 AND NOT #faultTrigg AND #iniOk AND (#laserModeM OR (#lasersOn AND #laserModeA));
END_REGION

REGION Network 6: включение группы лазеров
   RUNG wire#powerrail
      Contact( #enGreenUpLaser456 )
      I_Contact( #faultTrigg )
      Contact( #iniOk )
      wire#w1
      Contact( #laserModeM )
      wire#w2
      Coil( #greenUpLaser_456 )
   END_RUNG
   RUNG wire#w1
      Contact( #lasersOn )
      Contact( #laserModeA )
   END_RUNG wire#w2
   // the same network as SCL:
   #greenUpLaser_456 := #enGreenUpLaser456 AND NOT #faultTrigg AND #iniOk AND (#laserModeM OR (#lasersOn AND #laserModeA));
END_REGION

REGION Network 7: включение группы лазеров
   RUNG wire#powerrail
      Contact( #enBlueUpLaser789 )
      I_Contact( #faultTrigg )
      Contact( #iniOk )
      wire#w1
      Contact( #laserModeM )
      wire#w2
      Coil( #blueUpLaser_789 )
   END_RUNG
   RUNG wire#w1
      Contact( #lasersOn )
      Contact( #laserModeA )
   END_RUNG wire#w2
   // the same network as SCL:
   #blueUpLaser_789 := #enBlueUpLaser789 AND NOT #faultTrigg AND #iniOk AND (#laserModeM OR (#lasersOn AND #laserModeA));
END_REGION

REGION Network 8: включение группы лазеров
   RUNG wire#powerrail
      Contact( #enGreenDownLaser123 )
      I_Contact( #faultTrigg )
      Contact( #iniOk )
      wire#w1
      Contact( #laserModeM )
      wire#w2
      Coil( #greenDownLaser_123 )
   END_RUNG
   RUNG wire#w1
      Contact( #lasersOn )
      Contact( #laserModeA )
   END_RUNG wire#w2
   // the same network as SCL:
   #greenDownLaser_123 := #enGreenDownLaser123 AND NOT #faultTrigg AND #iniOk AND (#laserModeM OR (#lasersOn AND #laserModeA));
END_REGION

REGION Network 9: включение группы лазеров
   RUNG wire#powerrail
      Contact( #enBlueDownLaser123 )
      I_Contact( #faultTrigg )
      Contact( #iniOk )
      wire#w1
      Contact( #laserModeM )
      wire#w2
      Coil( #blueDownLaser_123 )
   END_RUNG
   RUNG wire#w1
      Contact( #lasersOn )
      Contact( #laserModeA )
   END_RUNG wire#w2
   // the same network as SCL:
   #blueDownLaser_123 := #enBlueDownLaser123 AND NOT #faultTrigg AND #iniOk AND (#laserModeM OR (#lasersOn AND #laserModeA));
END_REGION

REGION Network 10: включение группы лазеров
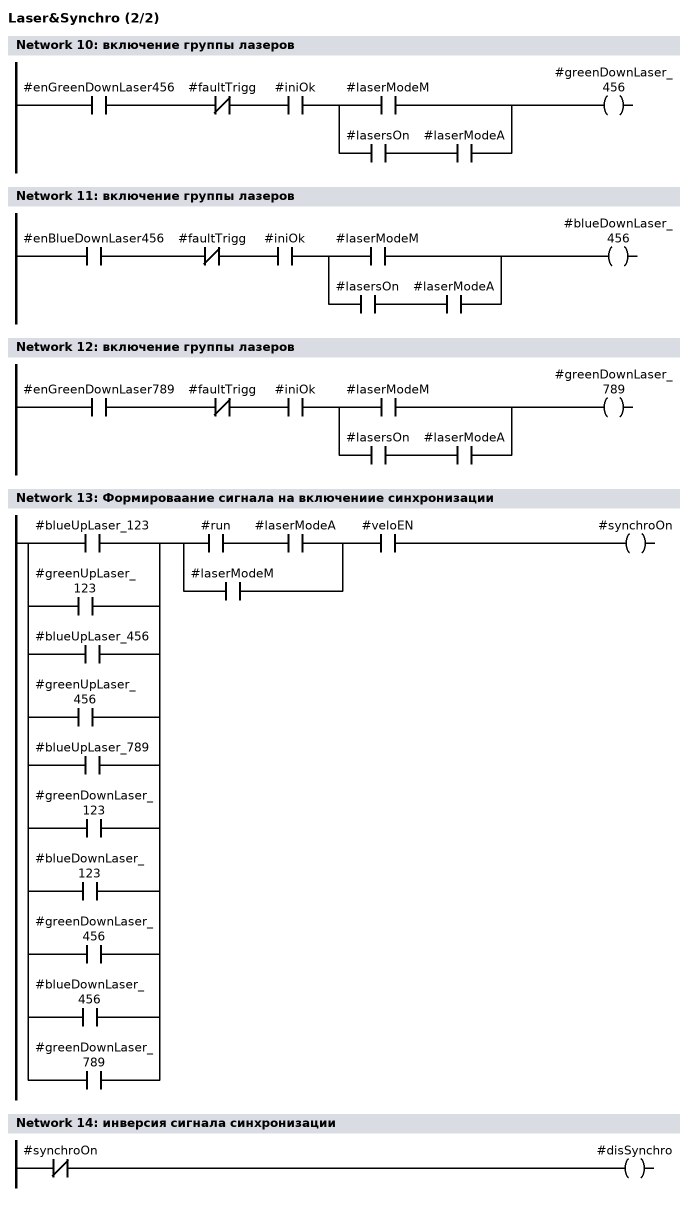
   RUNG wire#powerrail
      Contact( #enGreenDownLaser456 )
      I_Contact( #faultTrigg )
      Contact( #iniOk )
      wire#w1
      Contact( #laserModeM )
      wire#w2
      Coil( #greenDownLaser_456 )
   END_RUNG
   RUNG wire#w1
      Contact( #lasersOn )
      Contact( #laserModeA )
   END_RUNG wire#w2
   // the same network as SCL:
   #greenDownLaser_456 := #enGreenDownLaser456 AND NOT #faultTrigg AND #iniOk AND (#laserModeM OR (#lasersOn AND #laserModeA));
END_REGION

REGION Network 11: включение группы лазеров
   RUNG wire#powerrail
      Contact( #enBlueDownLaser456 )
      I_Contact( #faultTrigg )
      Contact( #iniOk )
      wire#w1
      Contact( #laserModeM )
      wire#w2
      Coil( #blueDownLaser_456 )
   END_RUNG
   RUNG wire#w1
      Contact( #lasersOn )
      Contact( #laserModeA )
   END_RUNG wire#w2
   // the same network as SCL:
   #blueDownLaser_456 := #enBlueDownLaser456 AND NOT #faultTrigg AND #iniOk AND (#laserModeM OR (#lasersOn AND #laserModeA));
END_REGION

REGION Network 12: включение группы лазеров
   RUNG wire#powerrail
      Contact( #enGreenDownLaser789 )
      I_Contact( #faultTrigg )
      Contact( #iniOk )
      wire#w1
      Contact( #laserModeM )
      wire#w2
      Coil( #greenDownLaser_789 )
   END_RUNG
   RUNG wire#w1
      Contact( #lasersOn )
      Contact( #laserModeA )
   END_RUNG wire#w2
   // the same network as SCL:
   #greenDownLaser_789 := #enGreenDownLaser789 AND NOT #faultTrigg AND #iniOk AND (#laserModeM OR (#lasersOn AND #laserModeA));
END_REGION

REGION Network 13: Формироваание сигнала на включениие синхронизации
   RUNG wire#powerrail
      Contact( #blueUpLaser_123 )
      wire#w1
      Contact( #run )
      Contact( #laserModeA )
      wire#w2
      Contact( #veloEN )
      Coil( #synchroOn )
   END_RUNG
   RUNG wire#powerrail
      Contact( #greenUpLaser_123 )
   END_RUNG wire#w1
   RUNG wire#powerrail
      Contact( #blueUpLaser_456 )
   END_RUNG wire#w1
   RUNG wire#powerrail
      Contact( #greenUpLaser_456 )
   END_RUNG wire#w1
   RUNG wire#powerrail
      Contact( #blueUpLaser_789 )
   END_RUNG wire#w1
   RUNG wire#powerrail
      Contact( #greenDownLaser_123 )
   END_RUNG wire#w1
   RUNG wire#powerrail
      Contact( #blueDownLaser_123 )
   END_RUNG wire#w1
   RUNG wire#powerrail
      Contact( #greenDownLaser_456 )
   END_RUNG wire#w1
   RUNG wire#powerrail
      Contact( #blueDownLaser_456 )
   END_RUNG wire#w1
   RUNG wire#powerrail
      Contact( #greenDownLaser_789 )
   END_RUNG wire#w1
   RUNG wire#w1
      Contact( #laserModeM )
   END_RUNG wire#w2
   // the same network as SCL:
   #synchroOn := (#blueUpLaser_123 OR #greenUpLaser_123 OR #blueUpLaser_456 OR #greenUpLaser_456 OR #blueUpLaser_789 OR #greenDownLaser_123 OR #blueDownLaser_123 OR #greenDownLaser_456 OR #blueDownLaser_456 OR #greenDownLaser_789) AND ((#run AND #laserModeA) OR #laserModeM) AND #veloEN;
END_REGION

REGION Network 14: инверсия сигнала синхронизации
   RUNG wire#powerrail
      I_Contact( #synchroOn )
      Coil( #disSynchro )
   END_RUNG
   // the same network as SCL:
   #disSynchro := NOT #synchroOn;
END_REGION
END_FUNCTION_BLOCK

FUNCTION_BLOCK "Outputs_Handler"   // FB16, LAD
{ S7_Optimized_Access := 'TRUE' }
VERSION : 0.1
   VAR
      ChangeReal_Instance : "ChangeReal";
   END_VAR
   VAR_TEMP
      valChanged : Bool;
   END_VAR
   VAR_TEMP   // added for the SCL form of the ladder/FBD networks
      _w1 : Bool;
   END_VAR
BEGIN

REGION Network 1: ловля изменение числа, чтобы записать сразу все лазеры
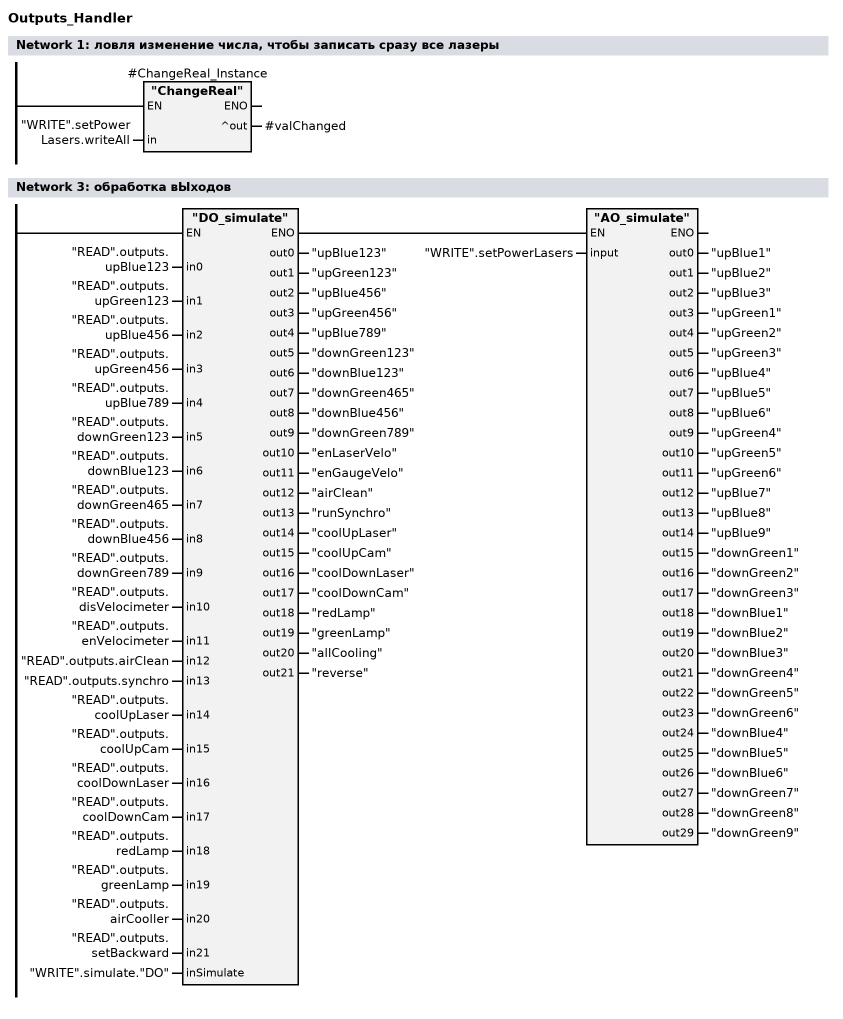
   RUNG wire#powerrail
      #ChangeReal_Instance(in := "WRITE".setPowerLasers.writeAll, "^out" => #valChanged)
   END_RUNG
   // the same network as SCL:
   #ChangeReal_Instance(in := "WRITE".setPowerLasers.writeAll, "^out" => #valChanged);   // "ChangeReal"
END_REGION

REGION Network 2 (SCL): Запись сразу всех значений мощности лазеров
   IF #valChanged THEN
       "WRITE".setPowerLasers.upBlue1 := "WRITE".setPowerLasers.writeAll;
       "WRITE".setPowerLasers.upBlue2 := "WRITE".setPowerLasers.writeAll;
       "WRITE".setPowerLasers.upBlue3 := "WRITE".setPowerLasers.writeAll;
       "WRITE".setPowerLasers.upGreen1 := "WRITE".setPowerLasers.writeAll;
       "WRITE".setPowerLasers.upGreen2 := "WRITE".setPowerLasers.writeAll;
       "WRITE".setPowerLasers.upGreen3 := "WRITE".setPowerLasers.writeAll;
       "WRITE".setPowerLasers.upBlue4 := "WRITE".setPowerLasers.writeAll;
       "WRITE".setPowerLasers.upBlue5 := "WRITE".setPowerLasers.writeAll;
       "WRITE".setPowerLasers.upBlue6 := "WRITE".setPowerLasers.writeAll;
       "WRITE".setPowerLasers.upGreen4 := "WRITE".setPowerLasers.writeAll;
       "WRITE".setPowerLasers.upGreen5 := "WRITE".setPowerLasers.writeAll;
       "WRITE".setPowerLasers.upGreen6 := "WRITE".setPowerLasers.writeAll;
       "WRITE".setPowerLasers.upBlue7 := "WRITE".setPowerLasers.writeAll;
       "WRITE".setPowerLasers.upBlue8 := "WRITE".setPowerLasers.writeAll;
       "WRITE".setPowerLasers.upBlue9 := "WRITE".setPowerLasers.writeAll;
       "WRITE".setPowerLasers.downGreen1 := "WRITE".setPowerLasers.writeAll;
       "WRITE".setPowerLasers.downGreen2 := "WRITE".setPowerLasers.writeAll;
       "WRITE".setPowerLasers.downGreen3 := "WRITE".setPowerLasers.writeAll;
       "WRITE".setPowerLasers.downBlue1 := "WRITE".setPowerLasers.writeAll;
       "WRITE".setPowerLasers.downBlue2 := "WRITE".setPowerLasers.writeAll;
       "WRITE".setPowerLasers.downBlue3 := "WRITE".setPowerLasers.writeAll;
       "WRITE".setPowerLasers.downGreen4 := "WRITE".setPowerLasers.writeAll;
       "WRITE".setPowerLasers.downGreen5 := "WRITE".setPowerLasers.writeAll;
       "WRITE".setPowerLasers.downGreen6 := "WRITE".setPowerLasers.writeAll;
       "WRITE".setPowerLasers.downBlue4 := "WRITE".setPowerLasers.writeAll;
       "WRITE".setPowerLasers.downBlue5 := "WRITE".setPowerLasers.writeAll;
       "WRITE".setPowerLasers.downBlue6 := "WRITE".setPowerLasers.writeAll;
       "WRITE".setPowerLasers.downGreen7 := "WRITE".setPowerLasers.writeAll;
       "WRITE".setPowerLasers.downGreen8 := "WRITE".setPowerLasers.writeAll;
       "WRITE".setPowerLasers.downGreen9 := "WRITE".setPowerLasers.writeAll;
   END_IF;
END_REGION

REGION Network 3: обработка вЫходов
   RUNG wire#powerrail
      "DO_simulate"(in0 := "READ".outputs.upBlue123, in1 := "READ".outputs.upGreen123, in2 := "READ".outputs.upBlue456, in3 := "READ".outputs.upGreen456, in4 := "READ".outputs.upBlue789, in5 := "READ".outputs.downGreen123, in6 := "READ".outputs.downBlue123, in7 := "READ".outputs.downGreen465, in8 := "READ".outputs.downBlue456, in9 := "READ".outputs.downGreen789, in10 := "READ".outputs.disVelocimeter, in11 := "READ".outputs.enVelocimeter, in12 := "READ".outputs.airClean, in13 := "READ".outputs.synchro, in14 := "READ".outputs.coolUpLaser, in15 := "READ".outputs.coolUpCam, in16 := "READ".outputs.coolDownLaser, in17 := "READ".outputs.coolDownCam, in18 := "READ".outputs.redLamp, in19 := "READ".outputs.greenLamp, in20 := "READ".outputs.airCooller, in21 := "READ".outputs.setBackward, inSimulate := "WRITE".simulate."DO", out0 => "upBlue123", out1 => "upGreen123", out2 => "upBlue456", out3 => "upGreen456", out4 => "upBlue789", out5 => "downGreen123", out6 => "downBlue123", out7 => "downGreen465", out8 => "downBlue456", out9 => "downGreen789", out10 => "enLaserVelo", out11 => "enGaugeVelo", out12 => "airClean", out13 => "runSynchro", out14 => "coolUpLaser", out15 => "coolUpCam", out16 => "coolDownLaser", out17 => "coolDownCam", out18 => "redLamp", out19 => "greenLamp", out20 => "allCooling", out21 => "reverse")
      "AO_simulate"(input := "WRITE".setPowerLasers, out0 => "upBlue1", out1 => "upBlue2", out2 => "upBlue3", out3 => "upGreen1", out4 => "upGreen2", out5 => "upGreen3", out6 => "upBlue4", out7 => "upBlue5", out8 => "upBlue6", out9 => "upGreen4", out10 => "upGreen5", out11 => "upGreen6", out12 => "upBlue7", out13 => "upBlue8", out14 => "upBlue9", out15 => "downGreen1", out16 => "downGreen2", out17 => "downGreen3", out18 => "downBlue1", out19 => "downBlue2", out20 => "downBlue3", out21 => "downGreen4", out22 => "downGreen5", out23 => "downGreen6", out24 => "downBlue4", out25 => "downBlue5", out26 => "downBlue6", out27 => "downGreen7", out28 => "downGreen8", out29 => "downGreen9")
   END_RUNG
   // the same network as SCL:
   "DO_simulate"(in0 := "READ".outputs.upBlue123,
                 in1 := "READ".outputs.upGreen123,
                 in2 := "READ".outputs.upBlue456,
                 in3 := "READ".outputs.upGreen456,
                 in4 := "READ".outputs.upBlue789,
                 in5 := "READ".outputs.downGreen123,
                 in6 := "READ".outputs.downBlue123,
                 in7 := "READ".outputs.downGreen465,
                 in8 := "READ".outputs.downBlue456,
                 in9 := "READ".outputs.downGreen789,
                 in10 := "READ".outputs.disVelocimeter,
                 in11 := "READ".outputs.enVelocimeter,
                 in12 := "READ".outputs.airClean,
                 in13 := "READ".outputs.synchro,
                 in14 := "READ".outputs.coolUpLaser,
                 in15 := "READ".outputs.coolUpCam,
                 in16 := "READ".outputs.coolDownLaser,
                 in17 := "READ".outputs.coolDownCam,
                 in18 := "READ".outputs.redLamp,
                 in19 := "READ".outputs.greenLamp,
                 in20 := "READ".outputs.airCooller,
                 in21 := "READ".outputs.setBackward,
                 inSimulate := "WRITE".simulate."DO",
                 out0 => "upBlue123",
                 out1 => "upGreen123",
                 out2 => "upBlue456",
                 out3 => "upGreen456",
                 out4 => "upBlue789",
                 out5 => "downGreen123",
                 out6 => "downBlue123",
                 out7 => "downGreen465",
                 out8 => "downBlue456",
                 out9 => "downGreen789",
                 out10 => "enLaserVelo",
                 out11 => "enGaugeVelo",
                 out12 => "airClean",
                 out13 => "runSynchro",
                 out14 => "coolUpLaser",
                 out15 => "coolUpCam",
                 out16 => "coolDownLaser",
                 out17 => "coolDownCam",
                 out18 => "redLamp",
                 out19 => "greenLamp",
                 out20 => "allCooling",
                 out21 => "reverse",
                 ENO => #_w1);
   IF #_w1 THEN
       "AO_simulate"(input := "WRITE".setPowerLasers,
                     out0 => "upBlue1",
                     out1 => "upBlue2",
                     out2 => "upBlue3",
                     out3 => "upGreen1",
                     out4 => "upGreen2",
                     out5 => "upGreen3",
                     out6 => "upBlue4",
                     out7 => "upBlue5",
                     out8 => "upBlue6",
                     out9 => "upGreen4",
                     out10 => "upGreen5",
                     out11 => "upGreen6",
                     out12 => "upBlue7",
                     out13 => "upBlue8",
                     out14 => "upBlue9",
                     out15 => "downGreen1",
                     out16 => "downGreen2",
                     out17 => "downGreen3",
                     out18 => "downBlue1",
                     out19 => "downBlue2",
                     out20 => "downBlue3",
                     out21 => "downGreen4",
                     out22 => "downGreen5",
                     out23 => "downGreen6",
                     out24 => "downBlue4",
                     out25 => "downBlue5",
                     out26 => "downBlue6",
                     out27 => "downGreen7",
                     out28 => "downGreen8",
                     out29 => "downGreen9");
   END_IF;
END_REGION
END_FUNCTION_BLOCK

ORGANIZATION_BLOCK "Main"   // OB1, LAD, ProgramCycle
TITLE = "Main Program Sweep (Cycle)"
{ S7_Optimized_Access := 'TRUE' }
VERSION : 0.1
   VAR_INPUT
      Initial_Call : Bool;   // Initial call of this OB
      Remanence : Bool;   // =True, if remanent data are available
   END_VAR
   VAR_TEMP
      iniAir : Bool;
      iniUpLaser : Bool;
      iniUpCam : Bool;
      iniDownLaser : Bool;
      iniDownCam : Bool;
      autoAir : Bool;
      autoUpLaser : Bool;
      autoUpCam : Bool;
      autoDownLaser : Bool;
      autoDownCam : Bool;
      synchro : Bool;
      tempNotAlarm : Bool;
   END_VAR
BEGIN

REGION Network 1: Обработка входов
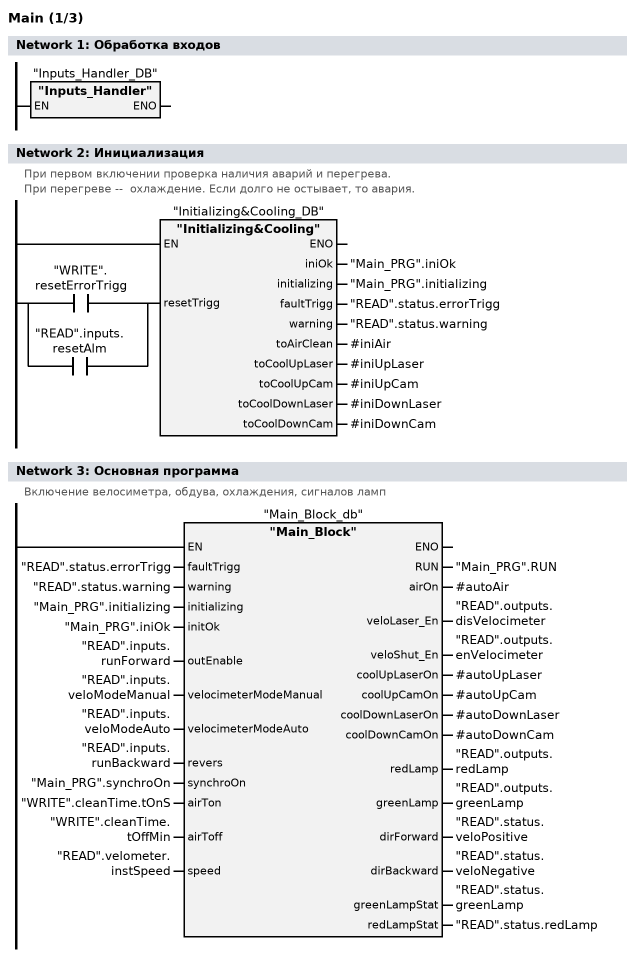
   RUNG wire#powerrail
      "Inputs_Handler_DB"()
   END_RUNG
   // the same network as SCL:
   "Inputs_Handler_DB"();   // "Inputs_Handler"
END_REGION

